LIN {X 0,Y 466.916,Z 269.289,A -85,B 0,C 180,E1 -7460.907,E2 -7460.907} C_VEL
LIN {X 0,Y 467.076,Z 265.162,A -85,B 0,C 180,E1 -7462.217,E2 -7462.217} C_VEL
LIN {X 0,Y 467.331,Z 259.259,A -85,B 0,C 180,E1 -7463.655,E2 -7463.655} C_VEL
LIN {X 0,Y 467.652,Z 252.016,A -85,B 0,C 180,E1 -7465.043,E2 -7465.043} C_VEL
LIN {X 0,Y 467.969,Z 245.037,A -85,B 0,C 180,E1 -7466.125,E2 -7466.125} C_VEL
LIN {X 0,Y 468.397,Z 236.625,A -85,B 0,C 180,E1 -7467.205,E2 -7467.205} C_VEL
LIN {X 0,Y 468.875,Z 226.254,A -85,B 0,C 180,E1 -7468.282,E2 -7468.282} C_VEL
LIN {X 0,Y 469.414,Z 214.581,A -85,B 0,C 180,E1 -7469.25,E2 -7469.25} C_VEL
LIN {X 0,Y 469.811,Z 202.915,A -85,B 0,C 180,E1 -7470,E2 -7470} C_VEL
LIN {X 0,Y 470.165,Z 189.535,A -85,B 0,C 180,E1 -7470.643,E2 -7470.643} C_VEL
LIN {X 0,Y 470.404,Z 177.571,A -85,B 0,C 180,E1 -7471.044,E2 -7471.044} C_VEL
LIN {X 0,Y 470.627,Z 162.533,A -85,B 0,C 180,E1 -7471.337,E2 -7471.337} C_VEL
LIN {X 0,Y 471.101,Z 78.839,A -85,B 0,C 180,E1 -7472.624,E2 -7472.624} C_VEL
LIN {X 0,Y 468.46,Z 65.811,A -85,B 0,C 180,E1 -7472.929,E2 -7472.929} C_VEL
LIN {X 0,Y 468.526,Z 59.499,A -85,B 0,C 180,E1 -7474.302,E2 -7474.302} C_VEL
LIN {X 0,Y 467.789,Z 54.217,A -85,B 0,C 180,E1 -7475.496,E2 -7475.496} C_VEL
LIN {X 0,Y 467.755,Z 54.218,A -85,B 0,C 180,E1 -7477.772,E2 -7477.772} C_VEL
LIN {X 0,Y 467.657,Z 54.228,A -85,B 0,C 180,E1 -7481.266,E2 -7481.266} C_VEL
LIN {X 0,Y 467.617,Z 54.234,A -85,B 0,C 180,E1 -7483.915,E2 -7483.915} C_VEL
LIN {X 0,Y 467.597,Z 54.24,A -85,B 0,C 180,E1 -7486.593,E2 -7486.593} C_VEL
LIN {X 0,Y 467.628,Z 54.231,A -85,B 0,C 180,E1 -7489.308,E2 -7489.308} C_VEL
LIN {X 0,Y 467.54,Z 54.248,A -85,B 0,C 180,E1 -7492.074,E2 -7492.074} C_VEL
LIN {X 0,Y 467.591,Z 54.236,A -85,B 0,C 180,E1 -7494.888,E2 -7494.888} C_VEL
LIN {X 0,Y 467.625,Z 54.236,A -85,B 0,C 180,E1 -7497.769,E2 -7497.769} C_VEL
LIN {X 0,Y 467.573,Z 54.238,A -85,B 0,C 180,E1 -7501.045,E2 -7501.045} C_VEL
LIN {X 0,Y 467.595,Z 54.237,A -85,B 0,C 180,E1 -7504.242,E2 -7504.242} C_VEL
LIN {X 0,Y 467.554,Z 54.242,A -85,B 0,C 180,E1 -7507.186,E2 -7507.186} C_VEL
LIN {X 0,Y 467.582,Z 54.237,A -85,B 0,C 180,E1 -7510.264,E2 -7510.264} C_VEL
LIN {X 0,Y 467.591,Z 54.236,A -85,B 0,C 180,E1 -7512.567,E2 -7512.567} C_VEL
LIN {X 0,Y 467.57,Z 54.242,A -85,B 0,C 180,E1 -7515.052,E2 -7515.052} C_VEL
LIN {X 0,Y 467.593,Z 54.241,A -85,B 0,C 180,E1 -7517.44,E2 -7517.44} C_VEL
LIN {X 0,Y 467.586,Z 54.24,A -85,B 0,C 180,E1 -7520.855,E2 -7520.855} C_VEL
LIN {X 0,Y 467.564,Z 54.239,A -85,B 0,C 180,E1 -7524.261,E2 -7524.261} C_VEL
LIN {X 0,Y 467.585,Z 54.239,A -85,B 0,C 180,E1 -7527.321,E2 -7527.321} C_VEL
LIN {X 0,Y 467.574,Z 54.244,A -85,B 0,C 180,E1 -7530.667,E2 -7530.667} C_VEL
LIN {X 0,Y 467.62,Z 54.234,A -85,B 0,C 180,E1 -7533.199,E2 -7533.199} C_VEL
LIN {X 0,Y 467.596,Z 54.241,A -85,B 0,C 180,E1 -7536.468,E2 -7536.468} C_VEL
LIN {X 0,Y 467.626,Z 54.232,A -85,B 0,C 180,E1 -7539.777,E2 -7539.777} C_VEL
LIN {X 0,Y 467.61,Z 54.24,A -85,B 0,C 180,E1 -7542.506,E2 -7542.506} C_VEL
LIN {X 0,Y 467.609,Z 54.233,A -85,B 0,C 180,E1 -7545.196,E2 -7545.196} C_VEL
LIN {X 0,Y 467.659,Z 54.23,A -85,B 0,C 180,E1 -7547.854,E2 -7547.854} C_VEL
LIN {X 0,Y 467.683,Z 54.225,A -85,B 0,C 180,E1 -7551.357,E2 -7551.357} C_VEL
LIN {X 0,Y 467.739,Z 54.225,A -85,B 0,C 180,E1 -7553.962,E2 -7553.962} C_VEL
LIN {X 0,Y 467.86,Z 54.204,A -85,B 0,C 180,E1 -7557.417,E2 -7557.417} C_VEL
LIN {X 0,Y 467.884,Z 54.204,A -85,B 0,C 180,E1 -7560,E2 -7560} C_VEL
LIN {X 0,Y 467.86,Z 54.202,A -85,B 0,C 180,E1 -7562.583,E2 -7562.583} C_VEL
LIN {X 0,Y 467.735,Z 54.22,A -85,B 0,C 180,E1 -7566.037,E2 -7566.037} C_VEL
LIN {X 0,Y 467.672,Z 54.226,A -85,B 0,C 180,E1 -7568.643,E2 -7568.643} C_VEL
LIN {X 0,Y 467.658,Z 54.227,A -85,B 0,C 180,E1 -7572.145,E2 -7572.145} C_VEL
LIN {X 0,Y 467.641,Z 54.232,A -85,B 0,C 180,E1 -7575.695,E2 -7575.695} C_VEL
LIN {X 0,Y 467.615,Z 54.236,A -85,B 0,C 180,E1 -7578.763,E2 -7578.763} C_VEL
LIN {X 0,Y 467.582,Z 54.241,A -85,B 0,C 180,E1 -7581.268,E2 -7581.268} C_VEL
LIN {X 0,Y 467.57,Z 54.238,A -85,B 0,C 180,E1 -7583.943,E2 -7583.943} C_VEL
LIN {X 0,Y 467.592,Z 54.243,A -85,B 0,C 180,E1 -7586.802,E2 -7586.802} C_VEL
LIN {X 0,Y 467.555,Z 54.24,A -85,B 0,C 180,E1 -7589.738,E2 -7589.738} C_VEL
LIN {X 0,Y 467.585,Z 54.243,A -85,B 0,C 180,E1 -7592.758,E2 -7592.758} C_VEL
LIN {X 0,Y 467.555,Z 54.241,A -85,B 0,C 180,E1 -7595.889,E2 -7595.889} C_VEL
LIN {X 0,Y 467.562,Z 54.24,A -85,B 0,C 180,E1 -7599.147,E2 -7599.147} C_VEL
LIN {X 0,Y 467.588,Z 54.24,A -85,B 0,C 180,E1 -7602.567,E2 -7602.567} C_VEL
LIN {X 0,Y 467.568,Z 54.239,A -85,B 0,C 180,E1 -7605.052,E2 -7605.052} C_VEL
LIN {X 0,Y 467.591,Z 54.236,A -85,B 0,C 180,E1 -7607.44,E2 -7607.44} C_VEL
LIN {X 0,Y 467.584,Z 54.237,A -85,B 0,C 180,E1 -7610.855,E2 -7610.855} C_VEL
LIN {X 0,Y 467.562,Z 54.242,A -85,B 0,C 180,E1 -7614.261,E2 -7614.261} C_VEL
LIN {X 0,Y 467.584,Z 54.239,A -85,B 0,C 180,E1 -7617.321,E2 -7617.321} C_VEL
LIN {X 0,Y 467.572,Z 54.244,A -85,B 0,C 180,E1 -7620.667,E2 -7620.667} C_VEL
LIN {X 0,Y 467.676,Z 54.389,A -85,B 0,C 180,E1 -7623.354,E2 -7623.354} C_VEL
LIN {X 0,Y 469.823,Z 66.098,A -85,B 0,C 180,E1 -7625.425,E2 -7625.425} C_VEL
LIN {X 0,Y 469.23,Z 83.836,A -85,B 0,C 180,E1 -7628.347,E2 -7628.347} C_VEL
LIN {X 0,Y 468.388,Z 105.455,A -85,B 0,C 180,E1 -7631.859,E2 -7631.859} C_VEL
LIN {X 0,Y 468.15,Z 113.126,A -85,B 0,C 180,E1 -7633.08,E2 -7633.08} C_VEL
LIN {X 0,Y 470.944,Z 133.853,A -85,B 0,C 180,E1 -7633.492,E2 -7633.492} C_VEL
LIN {X 0,Y 470.258,Z 222.266,A -85,B 0,C 180,E1 -7634.866,E2 -7634.866} C_VEL
LIN {X 0,Y 469.891,Z 235.42,A -85,B 0,C 180,E1 -7635.242,E2 -7635.242} C_VEL
LIN {X 0,Y 469.45,Z 247.547,A -85,B 0,C 180,E1 -7635.754,E2 -7635.754} C_VEL
LIN {X 0,Y 468.991,Z 259.804,A -85,B 0,C 180,E1 -7636.458,E2 -7636.458} C_VEL
LIN {X 0,Y 468.419,Z 272.106,A -85,B 0,C 180,E1 -7637.382,E2 -7637.382} C_VEL
LIN {X 0,Y 467.948,Z 282.93,A -85,B 0,C 180,E1 -7638.412,E2 -7638.412} C_VEL
LIN {X 0,Y 467.455,Z 292.948,A -85,B 0,C 180,E1 -7639.606,E2 -7639.606} C_VEL
LIN {X 0,Y 467.129,Z 301.775,A -85,B 0,C 180,E1 -7640.91,E2 -7640.91} C_VEL
LIN {X 0,Y 466.89,Z 308.811,A -85,B 0,C 180,E1 -7642.214,E2 -7642.214} C_VEL
LIN {X 0,Y 466.702,Z 314.993,A -85,B 0,C 180,E1 -7643.661,E2 -7643.661} C_VEL
LIN {X 0,Y 466.746,Z 318.872,A -85,B 0,C 180,E1 -7644.816,E2 -7644.816} C_VEL
LIN {X 0,Y 466.659,Z 321.204,A -85,B 0,C 180,E1 -7645.681,E2 -7645.681} C_VEL
LIN {X 0,Y 466.747,Z 323.112,A -85,B 0,C 180,E1 -7646.547,E2 -7646.547} C_VEL
LIN {X 0,Y 466.71,Z 324.547,A -85,B 0,C 180,E1 -7647.41,E2 -7647.41} C_VEL
LIN {X 0,Y 466.698,Z 325.564,A -85,B 0,C 180,E1 -7648.274,E2 -7648.274} C_VEL
LIN {X 0,Y 466.626,Z 326.421,A -85,B 0,C 180,E1 -7650,E2 -7650} C_VEL
LIN {X 0,Y 466.638,Z 326.228,A -85,B 0,C 180,E1 -7650.863,E2 -7650.863} C_VEL
LIN {X 0,Y 466.699,Z 325.63,A -85,B 0,C 180,E1 -7651.726,E2 -7651.726} C_VEL
LIN {X 0,Y 466.747,Z 323.253,A -85,B 0,C 180,E1 -7653.453,E2 -7653.453} C_VEL
LIN {X 0,Y 466.687,Z 320.32,A -85,B 0,C 180,E1 -7654.751,E2 -7654.751} C_VEL
LIN {X 0,Y 466.705,Z 316.357,A -85,B 0,C 180,E1 -7656.051,E2 -7656.051} C_VEL
LIN {X 0,Y 466.852,Z 311.265,A -85,B 0,C 180,E1 -7657.351,E2 -7657.351} C_VEL
LIN {X 0,Y 467.058,Z 304.877,A -85,B 0,C 180,E1 -7658.654,E2 -7658.654} C_VEL
LIN {X 0,Y 467.345,Z 296.895,A -85,B 0,C 180,E1 -7659.958,E2 -7659.958} C_VEL
LIN {X 0,Y 467.909,Z 286.997,A -85,B 0,C 180,E1 -7661.26,E2 -7661.26} C_VEL
LIN {X 0,Y 468.353,Z 277.342,A -85,B 0,C 180,E1 -7662.283,E2 -7662.283} C_VEL
LIN {X 0,Y 468.86,Z 266.461,A -85,B 0,C 180,E1 -7663.214,E2 -7663.214} C_VEL
LIN {X 0,Y 469.381,Z 255.345,A -85,B 0,C 180,E1 -7663.971,E2 -7663.971} C_VEL
LIN {X 0,Y 469.923,Z 243.021,A -85,B 0,C 180,E1 -7664.618,E2 -7664.618} C_VEL
LIN {X 0,Y 470.389,Z 229.964,A -85,B 0,C 180,E1 -7665.101,E2 -7665.101} C_VEL
LIN {X 0,Y 470.746,Z 217.491,A -85,B 0,C 180,E1 -7665.394,E2 -7665.394} C_VEL
LIN {X 0,Y 471.212,Z 132.613,A -85,B 0,C 180,E1 -7666.72,E2 -7666.72} C_VEL
LIN {X 0,Y 468.272,Z 112.505,A -85,B 0,C 180,E1 -7667.179,E2 -7667.179} C_VEL
LIN {X 0,Y 469.028,Z 94.371,A -85,B 0,C 180,E1 -7670.159,E2 -7670.159} C_VEL
LIN {X 0,Y 469.915,Z 73.905,A -85,B 0,C 180,E1 -7673.582,E2 -7673.582} C_VEL
LIN {X 0,Y 470.199,Z 67.087,A -85,B 0,C 180,E1 -7674.74,E2 -7674.74} C_VEL
LIN {X 0,Y 468.38,Z 57.447,A -85,B 0,C 180,E1 -7676.524,E2 -7676.524} C_VEL
LIN {X 0,Y 467.69,Z 54.229,A -85,B 0,C 180,E1 -7677.16,E2 -7677.16} C_VEL
LIN {X 0,Y 467.569,Z 54.245,A -85,B 0,C 180,E1 -7680.733,E2 -7680.733} C_VEL
LIN {X 0,Y 467.584,Z 54.244,A -85,B 0,C 180,E1 -7683.788,E2 -7683.788} C_VEL
LIN {X 0,Y 467.55,Z 54.243,A -85,B 0,C 180,E1 -7687.186,E2 -7687.186} C_VEL
LIN {X 0,Y 467.576,Z 54.242,A -85,B 0,C 180,E1 -7690.264,E2 -7690.264} C_VEL
LIN {X 0,Y 467.585,Z 54.238,A -85,B 0,C 180,E1 -7692.567,E2 -7692.567} C_VEL
LIN {X 0,Y 467.564,Z 54.239,A -85,B 0,C 180,E1 -7695.052,E2 -7695.052} C_VEL
LIN {X 0,Y 467.587,Z 54.241,A -85,B 0,C 180,E1 -7697.44,E2 -7697.44} C_VEL
LIN {X 0,Y 467.614,Z 54.235,A -85,B 0,C 180,E1 -7700.858,E2 -7700.858} C_VEL
LIN {X 0,Y 467.561,Z 54.24,A -85,B 0,C 180,E1 -7704.26,E2 -7704.26} C_VEL
LIN {X 0,Y 467.58,Z 54.243,A -85,B 0,C 180,E1 -7707.321,E2 -7707.321} C_VEL
LIN {X 0,Y 467.568,Z 54.242,A -85,B 0,C 180,E1 -7710.667,E2 -7710.667} C_VEL
LIN {X 0,Y 467.614,Z 54.234,A -85,B 0,C 180,E1 -7713.2,E2 -7713.2} C_VEL
LIN {X 0,Y 467.591,Z 54.241,A -85,B 0,C 180,E1 -7716.468,E2 -7716.468} C_VEL
LIN {X 0,Y 467.622,Z 54.233,A -85,B 0,C 180,E1 -7719.777,E2 -7719.777} C_VEL
LIN {X 0,Y 467.607,Z 54.235,A -85,B 0,C 180,E1 -7722.507,E2 -7722.507} C_VEL
LIN {X 0,Y 467.603,Z 54.235,A -85,B 0,C 180,E1 -7725.196,E2 -7725.196} C_VEL
LIN {X 0,Y 467.653,Z 54.225,A -85,B 0,C 180,E1 -7727.855,E2 -7727.855} C_VEL
LIN {X 0,Y 467.679,Z 54.224,A -85,B 0,C 180,E1 -7731.357,E2 -7731.357} C_VEL
LIN {X 0,Y 467.735,Z 54.222,A -85,B 0,C 180,E1 -7733.963,E2 -7733.963} C_VEL
LIN {X 0,Y 467.856,Z 54.203,A -85,B 0,C 180,E1 -7737.417,E2 -7737.417} C_VEL
LIN {X 0,Y 467.879,Z 54.205,A -85,B 0,C 180,E1 -7740,E2 -7740} C_VEL
LIN {X 0,Y 467.856,Z 54.198,A -85,B 0,C 180,E1 -7742.583,E2 -7742.583} C_VEL
LIN {X 0,Y 467.731,Z 54.22,A -85,B 0,C 180,E1 -7746.038,E2 -7746.038} C_VEL
LIN {X 0,Y 467.668,Z 54.222,A -85,B 0,C 180,E1 -7748.643,E2 -7748.643} C_VEL
LIN {X 0,Y 467.654,Z 54.226,A -85,B 0,C 180,E1 -7752.146,E2 -7752.146} C_VEL
LIN {X 0,Y 467.637,Z 54.231,A -85,B 0,C 180,E1 -7755.695,E2 -7755.695} C_VEL
LIN {X 0,Y 467.611,Z 54.236,A -85,B 0,C 180,E1 -7758.763,E2 -7758.763} C_VEL
LIN {X 0,Y 467.579,Z 54.236,A -85,B 0,C 180,E1 -7761.269,E2 -7761.269} C_VEL
LIN {X 0,Y 467.562,Z 54.241,A -85,B 0,C 180,E1 -7763.944,E2 -7763.944} C_VEL
LIN {X 0,Y 467.564,Z 54.245,A -85,B 0,C 180,E1 -7766.804,E2 -7766.804} C_VEL
LIN {X 0,Y 467.546,Z 54.24,A -85,B 0,C 180,E1 -7769.739,E2 -7769.739} C_VEL
LIN {X 0,Y 467.578,Z 54.241,A -85,B 0,C 180,E1 -7772.759,E2 -7772.759} C_VEL
LIN {X 0,Y 467.549,Z 54.243,A -85,B 0,C 180,E1 -7775.891,E2 -7775.891} C_VEL
LIN {X 0,Y 467.551,Z 54.244,A -85,B 0,C 180,E1 -7779.148,E2 -7779.148} C_VEL
LIN {X 0,Y 467.564,Z 54.237,A -85,B 0,C 180,E1 -7781.405,E2 -7781.405} C_VEL
LIN {X 0,Y 467.565,Z 54.239,A -85,B 0,C 180,E1 -7785.053,E2 -7785.053} C_VEL
LIN {X 0,Y 467.565,Z 54.24,A -85,B 0,C 180,E1 -7788.726,E2 -7788.726} C_VEL
LIN {X 0,Y 467.547,Z 54.248,A -85,B 0,C 180,E1 -7791.954,E2 -7791.954} C_VEL
LIN {X 0,Y 467.557,Z 54.249,A -85,B 0,C 180,E1 -7795.167,E2 -7795.167} C_VEL
LIN {X 0,Y 467.605,Z 54.347,A -85,B 0,C 180,E1 -7796.186,E2 -7796.186} C_VEL
LIN {X 0,Y 468.85,Z 61.426,A -85,B 0,C 180,E1 -7797.85,E2 -7797.85} C_VEL
LIN {X 0,Y 468.805,Z 66.288,A -85,B 0,C 180,E1 -7798.924,E2 -7798.924} C_VEL
LIN {X 0,Y 471.832,Z 79.918,A -85,B 0,C 180,E1 -7799.269,E2 -7799.269} C_VEL
LIN {X 0,Y 470.938,Z 172.284,A -85,B 0,C 180,E1 -7800.712,E2 -7800.712} C_VEL
LIN {X 0,Y 470.743,Z 183.575,A -85,B 0,C 180,E1 -7801.021,E2 -7801.021} C_VEL
LIN {X 0,Y 469.895,Z 189.287,A -85,B 0,C 180,E1 -7801.202,E2 -7801.202} C_VEL
LIN {X 0,Y 465.53,Z 201.989,A -85,B 0,C 180,E1 -7801.65,E2 -7801.65} C_VEL
LIN {X 0,Y 463.438,Z 209.017,A -85,B 0,C 180,E1 -7802.003,E2 -7802.003} C_VEL
LIN {X 0,Y 463.007,Z 212.433,A -85,B 0,C 180,E1 -7802.226,E2 -7802.226} C_VEL
LIN {X 0,Y 462.443,Z 223.732,A -85,B 0,C 180,E1 -7803.12,E2 -7803.12} C_VEL
LIN {X 0,Y 461.959,Z 233.267,A -85,B 0,C 180,E1 -7804.063,E2 -7804.063} C_VEL
LIN {X 0,Y 461.391,Z 242.873,A -85,B 0,C 180,E1 -7805.236,E2 -7805.236} C_VEL
LIN {X 0,Y 460.939,Z 250.637,A -85,B 0,C 180,E1 -7806.398,E2 -7806.398} C_VEL
LIN {X 0,Y 460.489,Z 258.274,A -85,B 0,C 180,E1 -7807.807,E2 -7807.807} C_VEL
LIN {X 0,Y 460.247,Z 263.603,A -85,B 0,C 180,E1 -7809.043,E2 -7809.043} C_VEL
LIN {X 0,Y 460.05,Z 268.129,A -85,B 0,C 180,E1 -7810.362,E2 -7810.362} C_VEL
LIN {X 0,Y 459.871,Z 270.811,A -85,B 0,C 180,E1 -7811.357,E2 -7811.357} C_VEL
LIN {X 0,Y 459.657,Z 274.227,A -85,B 0,C 180,E1 -7813.112,E2 -7813.112} C_VEL
LIN {X 0,Y 459.619,Z 275.682,A -85,B 0,C 180,E1 -7814.437,E2 -7814.437} C_VEL
LIN {X 0,Y 459.56,Z 276.252,A -85,B 0,C 180,E1 -7815.837,E2 -7815.837} C_VEL
LIN {X 0,Y 459.59,Z 276.094,A -85,B 0,C 180,E1 -7816.74,E2 -7816.74} C_VEL
LIN {X 0,Y 459.679,Z 275.066,A -85,B 0,C 180,E1 -7818.098,E2 -7818.098} C_VEL
LIN {X 0,Y 459.712,Z 273.122,A -85,B 0,C 180,E1 -7819.429,E2 -7819.429} C_VEL
LIN {X 0,Y 459.812,Z 270.194,A -85,B 0,C 180,E1 -7820.765,E2 -7820.765} C_VEL
LIN {X 0,Y 459.995,Z 266.224,A -85,B 0,C 180,E1 -7822.097,E2 -7822.097} C_VEL
LIN {X 0,Y 460.259,Z 260.296,A -85,B 0,C 180,E1 -7823.605,E2 -7823.605} C_VEL
LIN {X 0,Y 460.547,Z 253.46,A -85,B 0,C 180,E1 -7824.966,E2 -7824.966} C_VEL
LIN {X 0,Y 460.967,Z 245.209,A -85,B 0,C 180,E1 -7826.285,E2 -7826.285} C_VEL
LIN {X 0,Y 461.429,Z 236.726,A -85,B 0,C 180,E1 -7827.381,E2 -7827.381} C_VEL
LIN {X 0,Y 461.914,Z 226.288,A -85,B 0,C 180,E1 -7828.475,E2 -7828.475} C_VEL
LIN {X 0,Y 462.427,Z 215.936,A -85,B 0,C 180,E1 -7829.347,E2 -7829.347} C_VEL
LIN {X 0,Y 462.863,Z 204.608,A -85,B 0,C 180,E1 -7830.109,E2 -7830.109} C_VEL
LIN {X 0,Y 463.241,Z 191.654,A -85,B 0,C 180,E1 -7830.761,E2 -7830.761} C_VEL
LIN {X 0,Y 463.48,Z 179.532,A -85,B 0,C 180,E1 -7831.195,E2 -7831.195} C_VEL
LIN {X 0,Y 463.668,Z 166.043,A -85,B 0,C 180,E1 -7831.493,E2 -7831.493} C_VEL
LIN {X 0,Y 464.364,Z 80.659,A -85,B 0,C 180,E1 -7832.82,E2 -7832.82} C_VEL
LIN {X 0,Y 461.461,Z 66.202,A -85,B 0,C 180,E1 -7833.153,E2 -7833.153} C_VEL
LIN {X 0,Y 461.55,Z 60.66,A -85,B 0,C 180,E1 -7834.367,E2 -7834.367} C_VEL
LIN {X 0,Y 460.751,Z 55.093,A -85,B 0,C 180,E1 -7835.663,E2 -7835.663} C_VEL
LIN {X 0,Y 460.701,Z 55.098,A -85,B 0,C 180,E1 -7837.892,E2 -7837.892} C_VEL
LIN {X 0,Y 460.616,Z 55.104,A -85,B 0,C 180,E1 -7841.441,E2 -7841.441} C_VEL
LIN {X 0,Y 460.571,Z 55.111,A -85,B 0,C 180,E1 -7845.035,E2 -7845.035} C_VEL
LIN {X 0,Y 460.555,Z 55.114,A -85,B 0,C 180,E1 -7847.77,E2 -7847.77} C_VEL
LIN {X 0,Y 460.557,Z 55.116,A -85,B 0,C 180,E1 -7850.547,E2 -7850.547} C_VEL
LIN {X 0,Y 460.537,Z 55.117,A -85,B 0,C 180,E1 -7853.704,E2 -7853.704} C_VEL
LIN {X 0,Y 460.561,Z 55.116,A -85,B 0,C 180,E1 -7856.266,E2 -7856.266} C_VEL
LIN {X 0,Y 460.544,Z 55.114,A -85,B 0,C 180,E1 -7859.231,E2 -7859.231} C_VEL
LIN {X 0,Y 460.537,Z 55.117,A -85,B 0,C 180,E1 -7862.284,E2 -7862.284} C_VEL
LIN {X 0,Y 460.518,Z 55.121,A -85,B 0,C 180,E1 -7865.445,E2 -7865.445} C_VEL
LIN {X 0,Y 460.549,Z 55.114,A -85,B 0,C 180,E1 -7868.898,E2 -7868.898} C_VEL
LIN {X 0,Y 460.527,Z 55.116,A -85,B 0,C 180,E1 -7872.181,E2 -7872.181} C_VEL
LIN {X 0,Y 460.518,Z 55.124,A -85,B 0,C 180,E1 -7875.411,E2 -7875.411} C_VEL
LIN {X 0,Y 460.536,Z 55.115,A -85,B 0,C 180,E1 -7878.397,E2 -7878.397} C_VEL
LIN {X 0,Y 460.53,Z 55.121,A -85,B 0,C 180,E1 -7881.267,E2 -7881.267} C_VEL
LIN {X 0,Y 460.514,Z 55.119,A -85,B 0,C 180,E1 -7884.554,E2 -7884.554} C_VEL
LIN {X 0,Y 460.535,Z 55.115,A -85,B 0,C 180,E1 -7887.715,E2 -7887.715} C_VEL
LIN {X 0,Y 460.544,Z 55.121,A -85,B 0,C 180,E1 -7890.769,E2 -7890.769} C_VEL
LIN {X 0,Y 460.566,Z 55.111,A -85,B 0,C 180,E1 -7893.735,E2 -7893.735} C_VEL
LIN {X 0,Y 460.549,Z 55.121,A -85,B 0,C 180,E1 -7896.624,E2 -7896.624} C_VEL
LIN {X 0,Y 460.554,Z 55.112,A -85,B 0,C 180,E1 -7899.453,E2 -7899.453} C_VEL
LIN {X 0,Y 460.561,Z 55.117,A -85,B 0,C 180,E1 -7902.23,E2 -7902.23} C_VEL
LIN {X 0,Y 460.568,Z 55.111,A -85,B 0,C 180,E1 -7904.965,E2 -7904.965} C_VEL
LIN {X 0,Y 460.613,Z 55.108,A -85,B 0,C 180,E1 -7908.559,E2 -7908.559} C_VEL
LIN {X 0,Y 460.698,Z 55.102,A -85,B 0,C 180,E1 -7912.108,E2 -7912.108} C_VEL
LIN {X 0,Y 460.697,Z 55.095,A -85,B 0,C 180,E1 -7914.748,E2 -7914.748} C_VEL
LIN {X 0,Y 460.801,Z 55.083,A -85,B 0,C 180,E1 -7917.377,E2 -7917.377} C_VEL
LIN {X 0,Y 460.854,Z 55.08,A -85,B 0,C 180,E1 -7920,E2 -7920} C_VEL
LIN {X 0,Y 460.801,Z 55.081,A -85,B 0,C 180,E1 -7922.622,E2 -7922.622} C_VEL
LIN {X 0,Y 460.7,Z 55.095,A -85,B 0,C 180,E1 -7926.13,E2 -7926.13} C_VEL
LIN {X 0,Y 460.622,Z 55.104,A -85,B 0,C 180,E1 -7928.776,E2 -7928.776} C_VEL
LIN {X 0,Y 460.616,Z 55.104,A -85,B 0,C 180,E1 -7932.445,E2 -7932.445} C_VEL
LIN {X 0,Y 460.602,Z 55.106,A -85,B 0,C 180,E1 -7935.997,E2 -7935.997} C_VEL
LIN {X 0,Y 460.57,Z 55.112,A -85,B 0,C 180,E1 -7939.615,E2 -7939.615} C_VEL
LIN {X 0,Y 460.512,Z 55.119,A -85,B 0,C 180,E1 -7942.429,E2 -7942.429} C_VEL
LIN {X 0,Y 460.55,Z 55.113,A -85,B 0,C 180,E1 -7945.797,E2 -7945.797} C_VEL
LIN {X 0,Y 460.551,Z 55.114,A -85,B 0,C 180,E1 -7948.233,E2 -7948.233} C_VEL
LIN {X 0,Y 460.523,Z 55.117,A -85,B 0,C 180,E1 -7951.283,E2 -7951.283} C_VEL
LIN {X 0,Y 460.533,Z 55.122,A -85,B 0,C 180,E1 -7954.505,E2 -7954.505} C_VEL
LIN {X 0,Y 460.503,Z 55.119,A -85,B 0,C 180,E1 -7957.623,E2 -7957.623} C_VEL
LIN {X 0,Y 460.541,Z 55.12,A -85,B 0,C 180,E1 -7960.269,E2 -7960.269} C_VEL
LIN {X 0,Y 460.498,Z 55.119,A -85,B 0,C 180,E1 -7963.376,E2 -7963.376} C_VEL
LIN {X 0,Y 460.498,Z 55.121,A -85,B 0,C 180,E1 -7966.624,E2 -7966.624} C_VEL
LIN {X 0,Y 460.544,Z 55.117,A -85,B 0,C 180,E1 -7969.73,E2 -7969.73} C_VEL
LIN {X 0,Y 460.501,Z 55.12,A -85,B 0,C 180,E1 -7972.524,E2 -7972.524} C_VEL
LIN {X 0,Y 460.549,Z 55.118,A -85,B 0,C 180,E1 -7975.624,E2 -7975.624} C_VEL
LIN {X 0,Y 460.539,Z 55.114,A -85,B 0,C 180,E1 -7978.744,E2 -7978.744} C_VEL
LIN {X 0,Y 460.584,Z 55.116,A -85,B 0,C 180,E1 -7982.254,E2 -7982.254} C_VEL
LIN {X 0,Y 460.642,Z 55.195,A -85,B 0,C 180,E1 -7983.159,E2 -7983.159} C_VEL
LIN {X 0,Y 462.889,Z 67.415,A -85,B 0,C 180,E1 -7985.356,E2 -7985.356} C_VEL
LIN {X 0,Y 462.112,Z 86.808,A -85,B 0,C 180,E1 -7988.592,E2 -7988.592} C_VEL
LIN {X 0,Y 461.363,Z 106.289,A -85,B 0,C 180,E1 -7991.803,E2 -7991.803} C_VEL
LIN {X 0,Y 461.13,Z 112.601,A -85,B 0,C 180,E1 -7992.836,E2 -7992.836} C_VEL
LIN {X 0,Y 464.07,Z 135.367,A -85,B 0,C 180,E1 -7993.297,E2 -7993.297} C_VEL
LIN {X 0,Y 463.357,Z 221.938,A -85,B 0,C 180,E1 -7994.663,E2 -7994.663} C_VEL
LIN {X 0,Y 462.977,Z 235.088,A -85,B 0,C 180,E1 -7995.045,E2 -7995.045} C_VEL
LIN {X 0,Y 462.496,Z 247.782,A -85,B 0,C 180,E1 -7995.591,E2 -7995.591} C_VEL
LIN {X 0,Y 462.028,Z 259.069,A -85,B 0,C 180,E1 -7996.25,E2 -7996.25} C_VEL
LIN {X 0,Y 461.496,Z 270.047,A -85,B 0,C 180,E1 -7997.069,E2 -7997.069} C_VEL
LIN {X 0,Y 460.94,Z 281.29,A -85,B 0,C 180,E1 -7998.121,E2 -7998.121} C_VEL
LIN {X 0,Y 460.544,Z 290.756,A -85,B 0,C 180,E1 -7999.226,E2 -7999.226} C_VEL
LIN {X 0,Y 460.118,Z 299.888,A -85,B 0,C 180,E1 -8000.549,E2 -8000.549} C_VEL
LIN {X 0,Y 459.884,Z 307.251,A -85,B 0,C 180,E1 -8001.873,E2 -8001.873} C_VEL
LIN {X 0,Y 459.733,Z 312.232,A -85,B 0,C 180,E1 -8002.975,E2 -8002.975} C_VEL
LIN {X 0,Y 459.621,Z 317.066,A -85,B 0,C 180,E1 -8004.296,E2 -8004.296} C_VEL
LIN {X 0,Y 459.574,Z 320.767,A -85,B 0,C 180,E1 -8005.614,E2 -8005.614} C_VEL
LIN {X 0,Y 459.657,Z 322.684,A -85,B 0,C 180,E1 -8006.493,E2 -8006.493} C_VEL
LIN {X 0,Y 459.631,Z 324.136,A -85,B 0,C 180,E1 -8007.371,E2 -8007.371} C_VEL
LIN {X 0,Y 459.635,Z 325.162,A -85,B 0,C 180,E1 -8008.247,E2 -8008.247} C_VEL
LIN {X 0,Y 459.556,Z 326.034,A -85,B 0,C 180,E1 -8010,E2 -8010} C_VEL
LIN {X 0,Y 459.57,Z 325.856,A -85,B 0,C 180,E1 -8010.876,E2 -8010.876} C_VEL
LIN {X 0,Y 459.606,Z 325.264,A -85,B 0,C 180,E1 -8011.752,E2 -8011.752} C_VEL
LIN {X 0,Y 459.63,Z 324.281,A -85,B 0,C 180,E1 -8012.629,E2 -8012.629} C_VEL
LIN {X 0,Y 459.64,Z 322.9,A -85,B 0,C 180,E1 -8013.506,E2 -8013.506} C_VEL
LIN {X 0,Y 459.613,Z 319.983,A -85,B 0,C 180,E1 -8014.824,E2 -8014.824} C_VEL
LIN {X 0,Y 459.634,Z 315.362,A -85,B 0,C 180,E1 -8016.342,E2 -8016.342} C_VEL
LIN {X 0,Y 459.861,Z 308.974,A -85,B 0,C 180,E1 -8017.906,E2 -8017.906} C_VEL
LIN {X 0,Y 460.066,Z 302.122,A -85,B 0,C 180,E1 -8019.23,E2 -8019.23} C_VEL
LIN {X 0,Y 460.468,Z 293.629,A -85,B 0,C 180,E1 -8020.553,E2 -8020.553} C_VEL
LIN {X 0,Y 460.98,Z 284.909,A -85,B 0,C 180,E1 -8021.654,E2 -8021.654} C_VEL
LIN {X 0,Y 461.531,Z 273.823,A -85,B 0,C 180,E1 -8022.791,E2 -8022.791} C_VEL
LIN {X 0,Y 462.121,Z 263.567,A -85,B 0,C 180,E1 -8023.634,E2 -8023.634} C_VEL
LIN {X 0,Y 462.661,Z 251.718,A -85,B 0,C 180,E1 -8024.403,E2 -8024.403} C_VEL
LIN {X 0,Y 463.252,Z 239.425,A -85,B 0,C 180,E1 -8025.002,E2 -8025.002} C_VEL
LIN {X 0,Y 463.731,Z 226.859,A -85,B 0,C 180,E1 -8025.436,E2 -8025.436} C_VEL
LIN {X 0,Y 463.962,Z 213.966,A -85,B 0,C 180,E1 -8025.71,E2 -8025.71} C_VEL
LIN {X 0,Y 464.636,Z 134.861,A -85,B 0,C 180,E1 -8026.951,E2 -8026.951} C_VEL
LIN {X 0,Y 461.857,Z 115.48,A -85,B 0,C 180,E1 -8027.38,E2 -8027.38} C_VEL
LIN {X 0,Y 461.325,Z 112.145,A -85,B 0,C 180,E1 -8027.471,E2 -8027.471} C_VEL
LIN {X 0,Y 462.091,Z 94.192,A -85,B 0,C 180,E1 -8030.475,E2 -8030.475} C_VEL
LIN {X 0,Y 463.114,Z 73.76,A -85,B 0,C 180,E1 -8033.95,E2 -8033.95} C_VEL
LIN {X 0,Y 463.247,Z 68.116,A -85,B 0,C 180,E1 -8034.933,E2 -8034.933} C_VEL
LIN {X 0,Y 460.815,Z 56.062,A -85,B 0,C 180,E1 -8037.228,E2 -8037.228} C_VEL
LIN {X 0,Y 460.625,Z 55.109,A -85,B 0,C 180,E1 -8037.449,E2 -8037.449} C_VEL
LIN {X 0,Y 460.511,Z 55.126,A -85,B 0,C 180,E1 -8040.24,E2 -8040.24} C_VEL
LIN {X 0,Y 460.527,Z 55.12,A -85,B 0,C 180,E1 -8043.325,E2 -8043.325} C_VEL
LIN {X 0,Y 460.478,Z 55.126,A -85,B 0,C 180,E1 -8046.529,E2 -8046.529} C_VEL
LIN {X 0,Y 460.557,Z 55.119,A -85,B 0,C 180,E1 -8049.859,E2 -8049.859} C_VEL
LIN {X 0,Y 460.511,Z 55.119,A -85,B 0,C 180,E1 -8052.9,E2 -8052.9} C_VEL
LIN {X 0,Y 460.507,Z 55.116,A -85,B 0,C 180,E1 -8055.83,E2 -8055.83} C_VEL
LIN {X 0,Y 460.537,Z 55.118,A -85,B 0,C 180,E1 -8058.989,E2 -8058.989} C_VEL
LIN {X 0,Y 460.542,Z 55.121,A -85,B 0,C 180,E1 -8061.269,E2 -8061.269} C_VEL
LIN {X 0,Y 460.512,Z 55.119,A -85,B 0,C 180,E1 -8064.554,E2 -8064.554} C_VEL
LIN {X 0,Y 460.529,Z 55.117,A -85,B 0,C 180,E1 -8067.715,E2 -8067.715} C_VEL
LIN {X 0,Y 460.538,Z 55.118,A -85,B 0,C 180,E1 -8070.769,E2 -8070.769} C_VEL
LIN {X 0,Y 460.561,Z 55.109,A -85,B 0,C 180,E1 -8073.735,E2 -8073.735} C_VEL
LIN {X 0,Y 460.544,Z 55.118,A -85,B 0,C 180,E1 -8076.624,E2 -8076.624} C_VEL
LIN {X 0,Y 460.55,Z 55.113,A -85,B 0,C 180,E1 -8079.453,E2 -8079.453} C_VEL
LIN {X 0,Y 460.557,Z 55.113,A -85,B 0,C 180,E1 -8082.23,E2 -8082.23} C_VEL
LIN {X 0,Y 460.563,Z 55.113,A -85,B 0,C 180,E1 -8084.965,E2 -8084.965} C_VEL
LIN {X 0,Y 460.609,Z 55.109,A -85,B 0,C 180,E1 -8088.559,E2 -8088.559} C_VEL
LIN {X 0,Y 460.693,Z 55.095,A -85,B 0,C 180,E1 -8092.109,E2 -8092.109} C_VEL
LIN {X 0,Y 460.693,Z 55.096,A -85,B 0,C 180,E1 -8094.748,E2 -8094.748} C_VEL
LIN {X 0,Y 460.797,Z 55.082,A -85,B 0,C 180,E1 -8097.378,E2 -8097.378} C_VEL
LIN {X 0,Y 460.849,Z 55.08,A -85,B 0,C 180,E1 -8100,E2 -8100} C_VEL
LIN {X 0,Y 460.797,Z 55.077,A -85,B 0,C 180,E1 -8102.623,E2 -8102.623} C_VEL
LIN {X 0,Y 460.696,Z 55.095,A -85,B 0,C 180,E1 -8106.13,E2 -8106.13} C_VEL
LIN {X 0,Y 460.618,Z 55.101,A -85,B 0,C 180,E1 -8108.777,E2 -8108.777} C_VEL
LIN {X 0,Y 460.611,Z 55.103,A -85,B 0,C 180,E1 -8112.445,E2 -8112.445} C_VEL
LIN {X 0,Y 460.598,Z 55.107,A -85,B 0,C 180,E1 -8115.998,E2 -8115.998} C_VEL
LIN {X 0,Y 460.566,Z 55.112,A -85,B 0,C 180,E1 -8119.616,E2 -8119.616} C_VEL
LIN {X 0,Y 460.509,Z 55.117,A -85,B 0,C 180,E1 -8122.429,E2 -8122.429} C_VEL
LIN {X 0,Y 460.547,Z 55.11,A -85,B 0,C 180,E1 -8125.797,E2 -8125.797} C_VEL
LIN {X 0,Y 460.525,Z 55.121,A -85,B 0,C 180,E1 -8128.235,E2 -8128.235} C_VEL
LIN {X 0,Y 460.519,Z 55.118,A -85,B 0,C 180,E1 -8131.283,E2 -8131.283} C_VEL
LIN {X 0,Y 460.521,Z 55.12,A -85,B 0,C 180,E1 -8134.504,E2 -8134.504} C_VEL
LIN {X 0,Y 460.497,Z 55.123,A -85,B 0,C 180,E1 -8137.624,E2 -8137.624} C_VEL
LIN {X 0,Y 460.518,Z 55.113,A -85,B 0,C 180,E1 -8141.013,E2 -8141.013} C_VEL
LIN {X 0,Y 460.511,Z 55.118,A -85,B 0,C 180,E1 -8144.59,E2 -8144.59} C_VEL
LIN {X 0,Y 460.491,Z 55.129,A -85,B 0,C 180,E1 -8147.816,E2 -8147.816} C_VEL
LIN {X 0,Y 460.511,Z 55.123,A -85,B 0,C 180,E1 -8150.136,E2 -8150.136} C_VEL
LIN {X 0,Y 460.467,Z 55.132,A -85,B 0,C 180,E1 -8153.47,E2 -8153.47} C_VEL
LIN {X 0,Y 460.562,Z 55.223,A -85,B 0,C 180,E1 -8155.956,E2 -8155.956} C_VEL
LIN {X 0,Y 461.93,Z 63.082,A -85,B 0,C 180,E1 -8157.826,E2 -8157.826} C_VEL
LIN {X 0,Y 461.938,Z 66.897,A -85,B 0,C 180,E1 -8158.63,E2 -8158.63} C_VEL
LIN {X 0,Y 465.085,Z 80.736,A -85,B 0,C 180,E1 -8158.995,E2 -8158.995} C_VEL
LIN {X 0,Y 464.185,Z 172.963,A -85,B 0,C 180,E1 -8160.462,E2 -8160.462} C_VEL
LIN {X 0,Y 463.93,Z 186.168,A -85,B 0,C 180,E1 -8160.848,E2 -8160.848} C_VEL
LIN {X 0,Y 463.585,Z 199.092,A -85,B 0,C 180,E1 -8161.414,E2 -8161.414} C_VEL
LIN {X 0,Y 463.133,Z 210.084,A -85,B 0,C 180,E1 -8162.062,E2 -8162.062} C_VEL
LIN {X 0,Y 463.007,Z 212.433,A -85,B 0,C 180,E1 -8162.226,E2 -8162.226} C_VEL
LIN {X 0,Y 462.15,Z 217.571,A -85,B 0,C 180,E1 -8162.581,E2 -8162.581} C_VEL
LIN {X 0,Y 458.965,Z 225.695,A -85,B 0,C 180,E1 -8163.173,E2 -8163.173} C_VEL
LIN {X 0,Y 455.745,Z 233.358,A -85,B 0,C 180,E1 -8163.842,E2 -8163.842} C_VEL
LIN {X 0,Y 454.807,Z 237.718,A -85,B 0,C 180,E1 -8164.322,E2 -8164.322} C_VEL
LIN {X 0,Y 454.29,Z 246.491,A -85,B 0,C 180,E1 -8165.503,E2 -8165.503} C_VEL
LIN {X 0,Y 453.784,Z 253.998,A -85,B 0,C 180,E1 -8166.739,E2 -8166.739} C_VEL
LIN {X 0,Y 453.351,Z 260.942,A -85,B 0,C 180,E1 -8168.158,E2 -8168.158} C_VEL
LIN {X 0,Y 453.11,Z 266.396,A -85,B 0,C 180,E1 -8169.575,E2 -8169.575} C_VEL
LIN {X 0,Y 452.827,Z 271.11,A -85,B 0,C 180,E1 -8171.217,E2 -8171.217} C_VEL
LIN {X 0,Y 452.596,Z 274.302,A -85,B 0,C 180,E1 -8172.841,E2 -8172.841} C_VEL
LIN {X 0,Y 452.529,Z 276.034,A -85,B 0,C 180,E1 -8174.344,E2 -8174.344} C_VEL
LIN {X 0,Y 452.489,Z 276.604,A -85,B 0,C 180,E1 -8175.611,E2 -8175.611} C_VEL
LIN {X 0,Y 452.485,Z 276.543,A -85,B 0,C 180,E1 -8176.528,E2 -8176.528} C_VEL
LIN {X 0,Y 452.589,Z 275.512,A -85,B 0,C 180,E1 -8178.042,E2 -8178.042} C_VEL
LIN {X 0,Y 452.637,Z 273.816,A -85,B 0,C 180,E1 -8179.262,E2 -8179.262} C_VEL
LIN {X 0,Y 452.721,Z 271.029,A -85,B 0,C 180,E1 -8180.619,E2 -8180.619} C_VEL
LIN {X 0,Y 452.907,Z 267.209,A -85,B 0,C 180,E1 -8181.972,E2 -8181.972} C_VEL
LIN {X 0,Y 453.121,Z 262.206,A -85,B 0,C 180,E1 -8183.336,E2 -8183.336} C_VEL
LIN {X 0,Y 453.427,Z 256.06,A -85,B 0,C 180,E1 -8184.664,E2 -8184.664} C_VEL
LIN {X 0,Y 453.785,Z 248.32,A -85,B 0,C 180,E1 -8186.004,E2 -8186.004} C_VEL
LIN {X 0,Y 454.337,Z 238.637,A -85,B 0,C 180,E1 -8187.341,E2 -8187.341} C_VEL
LIN {X 0,Y 454.877,Z 228.622,A -85,B 0,C 180,E1 -8188.451,E2 -8188.451} C_VEL
LIN {X 0,Y 455.438,Z 217.284,A -85,B 0,C 180,E1 -8189.448,E2 -8189.448} C_VEL
LIN {X 0,Y 455.909,Z 206.186,A -85,B 0,C 180,E1 -8190.221,E2 -8190.221} C_VEL
LIN {X 0,Y 456.27,Z 193.805,A -85,B 0,C 180,E1 -8190.883,E2 -8190.883} C_VEL
LIN {X 0,Y 456.569,Z 181.473,A -85,B 0,C 180,E1 -8191.351,E2 -8191.351} C_VEL
LIN {X 0,Y 456.782,Z 167.634,A -85,B 0,C 180,E1 -8191.681,E2 -8191.681} C_VEL
LIN {X 0,Y 457.471,Z 81.186,A -85,B 0,C 180,E1 -8193.046,E2 -8193.046} C_VEL
LIN {X 0,Y 454.529,Z 66.458,A -85,B 0,C 180,E1 -8193.408,E2 -8193.408} C_VEL
LIN {X 0,Y 454.568,Z 61.835,A -85,B 0,C 180,E1 -8194.434,E2 -8194.434} C_VEL
LIN {X 0,Y 453.71,Z 55.971,A -85,B 0,C 180,E1 -8195.835,E2 -8195.835} C_VEL
LIN {X 0,Y 453.658,Z 55.976,A -85,B 0,C 180,E1 -8198.015,E2 -8198.015} C_VEL
LIN {X 0,Y 453.565,Z 55.983,A -85,B 0,C 180,E1 -8201.621,E2 -8201.621} C_VEL
LIN {X 0,Y 453.546,Z 55.985,A -85,B 0,C 180,E1 -8205.274,E2 -8205.274} C_VEL
LIN {X 0,Y 453.51,Z 55.994,A -85,B 0,C 180,E1 -8208.056,E2 -8208.056} C_VEL
LIN {X 0,Y 453.488,Z 55.993,A -85,B 0,C 180,E1 -8210.882,E2 -8210.882} C_VEL
LIN {X 0,Y 453.5,Z 55.996,A -85,B 0,C 180,E1 -8213.887,E2 -8213.887} C_VEL
LIN {X 0,Y 453.507,Z 55.991,A -85,B 0,C 180,E1 -8216.706,E2 -8216.706} C_VEL
LIN {X 0,Y 453.48,Z 55.999,A -85,B 0,C 180,E1 -8219.732,E2 -8219.732} C_VEL
LIN {X 0,Y 453.496,Z 55.993,A -85,B 0,C 180,E1 -8223.189,E2 -8223.189} C_VEL
LIN {X 0,Y 453.46,Z 55.997,A -85,B 0,C 180,E1 -8226.299,E2 -8226.299} C_VEL
LIN {X 0,Y 453.521,Z 55.994,A -85,B 0,C 180,E1 -8229.447,E2 -8229.447} C_VEL
LIN {X 0,Y 453.467,Z 55.997,A -85,B 0,C 180,E1 -8232.995,E2 -8232.995} C_VEL
LIN {X 0,Y 453.467,Z 55.997,A -85,B 0,C 180,E1 -8235.779,E2 -8235.779} C_VEL
LIN {X 0,Y 453.483,Z 55.993,A -85,B 0,C 180,E1 -8238.209,E2 -8238.209} C_VEL
LIN {X 0,Y 453.498,Z 55.994,A -85,B 0,C 180,E1 -8240.793,E2 -8240.793} C_VEL
LIN {X 0,Y 453.458,Z 55.996,A -85,B 0,C 180,E1 -8243.917,E2 -8243.917} C_VEL
LIN {X 0,Y 453.486,Z 55.998,A -85,B 0,C 180,E1 -8247.151,E2 -8247.151} C_VEL
LIN {X 0,Y 453.478,Z 55.995,A -85,B 0,C 180,E1 -8250.268,E2 -8250.268} C_VEL
LIN {X 0,Y 453.51,Z 55.991,A -85,B 0,C 180,E1 -8253.294,E2 -8253.294} C_VEL
LIN {X 0,Y 453.507,Z 55.993,A -85,B 0,C 180,E1 -8256.239,E2 -8256.239} C_VEL
LIN {X 0,Y 453.485,Z 55.994,A -85,B 0,C 180,E1 -8259.117,E2 -8259.117} C_VEL
LIN {X 0,Y 453.514,Z 55.991,A -85,B 0,C 180,E1 -8261.944,E2 -8261.944} C_VEL
LIN {X 0,Y 453.543,Z 55.988,A -85,B 0,C 180,E1 -8264.726,E2 -8264.726} C_VEL
LIN {X 0,Y 453.562,Z 55.988,A -85,B 0,C 180,E1 -8268.379,E2 -8268.379} C_VEL
LIN {X 0,Y 453.655,Z 55.978,A -85,B 0,C 180,E1 -8271.985,E2 -8271.985} C_VEL
LIN {X 0,Y 453.67,Z 55.97,A -85,B 0,C 180,E1 -8274.667,E2 -8274.667} C_VEL
LIN {X 0,Y 453.745,Z 55.962,A -85,B 0,C 180,E1 -8277.336,E2 -8277.336} C_VEL
LIN {X 0,Y 453.824,Z 55.955,A -85,B 0,C 180,E1 -8280,E2 -8280} C_VEL
LIN {X 0,Y 453.745,Z 55.96,A -85,B 0,C 180,E1 -8282.663,E2 -8282.663} C_VEL
LIN {X 0,Y 453.668,Z 55.971,A -85,B 0,C 180,E1 -8286.225,E2 -8286.225} C_VEL
LIN {X 0,Y 453.588,Z 55.981,A -85,B 0,C 180,E1 -8288.913,E2 -8288.913} C_VEL
LIN {X 0,Y 453.566,Z 55.983,A -85,B 0,C 180,E1 -8292.529,E2 -8292.529} C_VEL
LIN {X 0,Y 453.546,Z 55.985,A -85,B 0,C 180,E1 -8296.196,E2 -8296.196} C_VEL
LIN {X 0,Y 453.519,Z 55.995,A -85,B 0,C 180,E1 -8299.039,E2 -8299.039} C_VEL
LIN {X 0,Y 453.478,Z 55.994,A -85,B 0,C 180,E1 -8301.836,E2 -8301.836} C_VEL
LIN {X 0,Y 453.505,Z 55.996,A -85,B 0,C 180,E1 -8304.735,E2 -8304.735} C_VEL
LIN {X 0,Y 453.53,Z 55.987,A -85,B 0,C 180,E1 -8307.959,E2 -8307.959} C_VEL
LIN {X 0,Y 453.467,Z 55.995,A -85,B 0,C 180,E1 -8311.525,E2 -8311.525} C_VEL
LIN {X 0,Y 453.489,Z 55.997,A -85,B 0,C 180,E1 -8314.777,E2 -8314.777} C_VEL
LIN {X 0,Y 453.462,Z 56.002,A -85,B 0,C 180,E1 -8318.312,E2 -8318.312} C_VEL
LIN {X 0,Y 453.495,Z 55.996,A -85,B 0,C 180,E1 -8320.609,E2 -8320.609} C_VEL
LIN {X 0,Y 453.454,Z 55.997,A -85,B 0,C 180,E1 -8323.244,E2 -8323.244} C_VEL
LIN {X 0,Y 453.464,Z 55.998,A -85,B 0,C 180,E1 -8325.778,E2 -8325.778} C_VEL
LIN {X 0,Y 453.481,Z 55.999,A -85,B 0,C 180,E1 -8328.209,E2 -8328.209} C_VEL
LIN {X 0,Y 453.496,Z 55.992,A -85,B 0,C 180,E1 -8330.793,E2 -8330.793} C_VEL
LIN {X 0,Y 453.457,Z 56.004,A -85,B 0,C 180,E1 -8333.917,E2 -8333.917} C_VEL
LIN {X 0,Y 453.485,Z 55.994,A -85,B 0,C 180,E1 -8337.151,E2 -8337.151} C_VEL
LIN {X 0,Y 453.477,Z 56.002,A -85,B 0,C 180,E1 -8340.268,E2 -8340.268} C_VEL
LIN {X 0,Y 453.614,Z 56.157,A -85,B 0,C 180,E1 -8342.99,E2 -8342.99} C_VEL
LIN {X 0,Y 455.856,Z 68.009,A -85,B 0,C 180,E1 -8345.158,E2 -8345.158} C_VEL
LIN {X 0,Y 455.465,Z 79.226,A -85,B 0,C 180,E1 -8347.069,E2 -8347.069} C_VEL
LIN {X 0,Y 454.746,Z 95.975,A -85,B 0,C 180,E1 -8349.887,E2 -8349.887} C_VEL
LIN {X 0,Y 454.114,Z 112.337,A -85,B 0,C 180,E1 -8352.604,E2 -8352.604} C_VEL
LIN {X 0,Y 457.214,Z 135.978,A -85,B 0,C 180,E1 -8353.086,E2 -8353.086} C_VEL
LIN {X 0,Y 456.457,Z 221.473,A -85,B 0,C 180,E1 -8354.454,E2 -8354.454} C_VEL
LIN {X 0,Y 456.066,Z 234.651,A -85,B 0,C 180,E1 -8354.841,E2 -8354.841} C_VEL
LIN {X 0,Y 455.58,Z 246.79,A -85,B 0,C 180,E1 -8355.368,E2 -8355.368} C_VEL
LIN {X 0,Y 455.07,Z 258.248,A -85,B 0,C 180,E1 -8356.036,E2 -8356.036} C_VEL
LIN {X 0,Y 454.506,Z 269.873,A -85,B 0,C 180,E1 -8356.915,E2 -8356.915} C_VEL
LIN {X 0,Y 453.943,Z 280.621,A -85,B 0,C 180,E1 -8357.935,E2 -8357.935} C_VEL
LIN {X 0,Y 453.53,Z 290.163,A -85,B 0,C 180,E1 -8359.057,E2 -8359.057} C_VEL
LIN {X 0,Y 453.073,Z 299.34,A -85,B 0,C 180,E1 -8360.401,E2 -8360.401} C_VEL
LIN {X 0,Y 452.813,Z 306.739,A -85,B 0,C 180,E1 -8361.745,E2 -8361.745} C_VEL
LIN {X 0,Y 452.657,Z 311.748,A -85,B 0,C 180,E1 -8362.865,E2 -8362.865} C_VEL
LIN {X 0,Y 452.525,Z 316.986,A -85,B 0,C 180,E1 -8364.324,E2 -8364.324} C_VEL
LIN {X 0,Y 452.494,Z 320.329,A -85,B 0,C 180,E1 -8365.546,E2 -8365.546} C_VEL
LIN {X 0,Y 452.553,Z 322.254,A -85,B 0,C 180,E1 -8366.438,E2 -8366.438} C_VEL
LIN {X 0,Y 452.553,Z 323.725,A -85,B 0,C 180,E1 -8367.329,E2 -8367.329} C_VEL
LIN {X 0,Y 452.543,Z 324.758,A -85,B 0,C 180,E1 -8368.22,E2 -8368.22} C_VEL
LIN {X 0,Y 452.488,Z 325.646,A -85,B 0,C 180,E1 -8370,E2 -8370} C_VEL
LIN {X 0,Y 452.504,Z 325.483,A -85,B 0,C 180,E1 -8370.89,E2 -8370.89} C_VEL
LIN {X 0,Y 452.552,Z 323.923,A -85,B 0,C 180,E1 -8372.67,E2 -8372.67} C_VEL
LIN {X 0,Y 452.536,Z 322.549,A -85,B 0,C 180,E1 -8373.561,E2 -8373.561} C_VEL
LIN {X 0,Y 452.539,Z 319.653,A -85,B 0,C 180,E1 -8374.9,E2 -8374.9} C_VEL
LIN {X 0,Y 452.553,Z 315.435,A -85,B 0,C 180,E1 -8376.331,E2 -8376.331} C_VEL
LIN {X 0,Y 452.719,Z 310.679,A -85,B 0,C 180,E1 -8377.582,E2 -8377.582} C_VEL
LIN {X 0,Y 452.923,Z 304.352,A -85,B 0,C 180,E1 -8378.926,E2 -8378.926} C_VEL
LIN {X 0,Y 453.281,Z 296.453,A -85,B 0,C 180,E1 -8380.271,E2 -8380.271} C_VEL
LIN {X 0,Y 453.83,Z 288.425,A -85,B 0,C 180,E1 -8381.387,E2 -8381.387} C_VEL
LIN {X 0,Y 454.327,Z 278.649,A -85,B 0,C 180,E1 -8382.507,E2 -8382.507} C_VEL
LIN {X 0,Y 454.935,Z 267.8,A -85,B 0,C 180,E1 -8383.512,E2 -8383.512} C_VEL
LIN {X 0,Y 455.536,Z 257.227,A -85,B 0,C 180,E1 -8384.291,E2 -8384.291} C_VEL
LIN {X 0,Y 456.19,Z 244.529,A -85,B 0,C 180,E1 -8385.011,E2 -8385.011} C_VEL
LIN {X 0,Y 456.699,Z 231.848,A -85,B 0,C 180,E1 -8385.537,E2 -8385.537} C_VEL
LIN {X 0,Y 457.161,Z 219.761,A -85,B 0,C 180,E1 -8385.864,E2 -8385.864} C_VEL
LIN {X 0,Y 457.76,Z 134.333,A -85,B 0,C 180,E1 -8387.249,E2 -8387.249} C_VEL
LIN {X 0,Y 454.779,Z 114.277,A -85,B 0,C 180,E1 -8387.71,E2 -8387.71} C_VEL
LIN {X 0,Y 454.366,Z 111.733,A -85,B 0,C 180,E1 -8387.784,E2 -8387.784} C_VEL
LIN {X 0,Y 455.142,Z 95.395,A -85,B 0,C 180,E1 -8390.566,E2 -8390.566} C_VEL
LIN {X 0,Y 456.237,Z 74.997,A -85,B 0,C 180,E1 -8394.092,E2 -8394.092} C_VEL
LIN {X 0,Y 456.352,Z 69.557,A -85,B 0,C 180,E1 -8395.056,E2 -8395.056} C_VEL
LIN {X 0,Y 453.901,Z 57.331,A -85,B 0,C 180,E1 -8397.428,E2 -8397.428} C_VEL
LIN {X 0,Y 453.546,Z 55.992,A -85,B 0,C 180,E1 -8397.701,E2 -8397.701} C_VEL
LIN {X 0,Y 453.476,Z 56,A -85,B 0,C 180,E1 -8400.759,E2 -8400.759} C_VEL
LIN {X 0,Y 453.476,Z 56.003,A -85,B 0,C 180,E1 -8403.912,E2 -8403.912} C_VEL
LIN {X 0,Y 453.47,Z 55.998,A -85,B 0,C 180,E1 -8407.187,E2 -8407.187} C_VEL
LIN {X 0,Y 453.516,Z 55.993,A -85,B 0,C 180,E1 -8409.447,E2 -8409.447} C_VEL
LIN {X 0,Y 453.461,Z 55.998,A -85,B 0,C 180,E1 -8412.995,E2 -8412.995} C_VEL
LIN {X 0,Y 453.462,Z 55.993,A -85,B 0,C 180,E1 -8415.778,E2 -8415.778} C_VEL
LIN {X 0,Y 453.514,Z 55.993,A -85,B 0,C 180,E1 -8419.405,E2 -8419.405} C_VEL
LIN {X 0,Y 453.475,Z 55.992,A -85,B 0,C 180,E1 -8422.222,E2 -8422.222} C_VEL
LIN {X 0,Y 453.487,Z 55.996,A -85,B 0,C 180,E1 -8425.222,E2 -8425.222} C_VEL
LIN {X 0,Y 453.464,Z 55.998,A -85,B 0,C 180,E1 -8428.475,E2 -8428.475} C_VEL
LIN {X 0,Y 453.535,Z 55.987,A -85,B 0,C 180,E1 -8432.039,E2 -8432.039} C_VEL
LIN {X 0,Y 453.512,Z 55.992,A -85,B 0,C 180,E1 -8435.266,E2 -8435.266} C_VEL
LIN {X 0,Y 453.478,Z 55.993,A -85,B 0,C 180,E1 -8438.415,E2 -8438.415} C_VEL
LIN {X 0,Y 453.52,Z 55.988,A -85,B 0,C 180,E1 -8441.009,E2 -8441.009} C_VEL
LIN {X 0,Y 453.566,Z 55.983,A -85,B 0,C 180,E1 -8443.88,E2 -8443.88} C_VEL
LIN {X 0,Y 453.561,Z 55.977,A -85,B 0,C 180,E1 -8447.471,E2 -8447.471} C_VEL
LIN {X 0,Y 453.59,Z 55.979,A -85,B 0,C 180,E1 -8451.087,E2 -8451.087} C_VEL
LIN {X 0,Y 453.669,Z 55.971,A -85,B 0,C 180,E1 -8453.775,E2 -8453.775} C_VEL
LIN {X 0,Y 453.741,Z 55.96,A -85,B 0,C 180,E1 -8457.337,E2 -8457.337} C_VEL
LIN {X 0,Y 453.82,Z 55.956,A -85,B 0,C 180,E1 -8460,E2 -8460} C_VEL
LIN {X 0,Y 453.741,Z 55.956,A -85,B 0,C 180,E1 -8462.664,E2 -8462.664} C_VEL
LIN {X 0,Y 453.663,Z 55.971,A -85,B 0,C 180,E1 -8466.226,E2 -8466.226} C_VEL
LIN {X 0,Y 453.584,Z 55.978,A -85,B 0,C 180,E1 -8468.914,E2 -8468.914} C_VEL
LIN {X 0,Y 453.561,Z 55.982,A -85,B 0,C 180,E1 -8472.529,E2 -8472.529} C_VEL
LIN {X 0,Y 453.542,Z 55.986,A -85,B 0,C 180,E1 -8476.196,E2 -8476.196} C_VEL
LIN {X 0,Y 453.516,Z 55.996,A -85,B 0,C 180,E1 -8479.04,E2 -8479.04} C_VEL
LIN {X 0,Y 453.475,Z 55.99,A -85,B 0,C 180,E1 -8481.837,E2 -8481.837} C_VEL
LIN {X 0,Y 453.5,Z 55.995,A -85,B 0,C 180,E1 -8484.736,E2 -8484.736} C_VEL
LIN {X 0,Y 453.505,Z 55.993,A -85,B 0,C 180,E1 -8487.954,E2 -8487.954} C_VEL
LIN {X 0,Y 453.474,Z 55.999,A -85,B 0,C 180,E1 -8490.76,E2 -8490.76} C_VEL
LIN {X 0,Y 453.467,Z 55.999,A -85,B 0,C 180,E1 -8493.914,E2 -8493.914} C_VEL
LIN {X 0,Y 453.448,Z 55.999,A -85,B 0,C 180,E1 -8497.191,E2 -8497.191} C_VEL
LIN {X 0,Y 453.47,Z 55.992,A -85,B 0,C 180,E1 -8500.612,E2 -8500.612} C_VEL
LIN {X 0,Y 453.459,Z 56,A -85,B 0,C 180,E1 -8504.223,E2 -8504.223} C_VEL
LIN {X 0,Y 453.437,Z 56.005,A -85,B 0,C 180,E1 -8507.003,E2 -8507.003} C_VEL
LIN {X 0,Y 453.471,Z 56.001,A -85,B 0,C 180,E1 -8509.413,E2 -8509.413} C_VEL
LIN {X 0,Y 453.44,Z 56.004,A -85,B 0,C 180,E1 -8512.81,E2 -8512.81} C_VEL
LIN {X 0,Y 453.532,Z 56.142,A -85,B 0,C 180,E1 -8515.724,E2 -8515.724} C_VEL
LIN {X 0,Y 455.012,Z 64.616,A -85,B 0,C 180,E1 -8517.772,E2 -8517.772} C_VEL
LIN {X 0,Y 455.028,Z 66.936,A -85,B 0,C 180,E1 -8518.303,E2 -8518.303} C_VEL
LIN {X 0,Y 458.344,Z 81.429,A -85,B 0,C 180,E1 -8518.705,E2 -8518.705} C_VEL
LIN {X 0,Y 457.444,Z 173.795,A -85,B 0,C 180,E1 -8520.204,E2 -8520.204} C_VEL
LIN {X 0,Y 457.18,Z 186.725,A -85,B 0,C 180,E1 -8520.592,E2 -8520.592} C_VEL
LIN {X 0,Y 456.827,Z 199.318,A -85,B 0,C 180,E1 -8521.153,E2 -8521.153} C_VEL
LIN {X 0,Y 456.283,Z 211.011,A -85,B 0,C 180,E1 -8521.855,E2 -8521.855} C_VEL
LIN {X 0,Y 455.713,Z 221.807,A -85,B 0,C 180,E1 -8522.69,E2 -8522.69} C_VEL
LIN {X 0,Y 455.137,Z 232.222,A -85,B 0,C 180,E1 -8523.696,E2 -8523.696} C_VEL
LIN {X 0,Y 454.807,Z 237.718,A -85,B 0,C 180,E1 -8524.322,E2 -8524.322} C_VEL
LIN {X 0,Y 453.881,Z 241.969,A -85,B 0,C 180,E1 -8524.828,E2 -8524.828} C_VEL
LIN {X 0,Y 450.642,Z 248.547,A -85,B 0,C 180,E1 -8525.676,E2 -8525.676} C_VEL
LIN {X 0,Y 447.45,Z 254.506,A -85,B 0,C 180,E1 -8526.602,E2 -8526.602} C_VEL
LIN {X 0,Y 446.609,Z 257.774,A -85,B 0,C 180,E1 -8527.223,E2 -8527.223} C_VEL
LIN {X 0,Y 446.209,Z 264.377,A -85,B 0,C 180,E1 -8528.761,E2 -8528.761} C_VEL
LIN {X 0,Y 445.96,Z 269.116,A -85,B 0,C 180,E1 -8530.195,E2 -8530.195} C_VEL
LIN {X 0,Y 445.676,Z 272.648,A -85,B 0,C 180,E1 -8531.616,E2 -8531.616} C_VEL
LIN {X 0,Y 445.539,Z 274.375,A -85,B 0,C 180,E1 -8532.56,E2 -8532.56} C_VEL
LIN {X 0,Y 445.444,Z 276.385,A -85,B 0,C 180,E1 -8534.246,E2 -8534.246} C_VEL
LIN {X 0,Y 445.406,Z 276.958,A -85,B 0,C 180,E1 -8535.377,E2 -8535.377} C_VEL
LIN {X 0,Y 445.407,Z 276.964,A -85,B 0,C 180,E1 -8536.31,E2 -8536.31} C_VEL
LIN {X 0,Y 445.512,Z 275.956,A -85,B 0,C 180,E1 -8537.978,E2 -8537.978} C_VEL
LIN {X 0,Y 445.548,Z 274.51,A -85,B 0,C 180,E1 -8539.089,E2 -8539.089} C_VEL
LIN {X 0,Y 445.638,Z 271.864,A -85,B 0,C 180,E1 -8540.469,E2 -8540.469} C_VEL
LIN {X 0,Y 445.821,Z 268.193,A -85,B 0,C 180,E1 -8541.844,E2 -8541.844} C_VEL
LIN {X 0,Y 446.052,Z 262.958,A -85,B 0,C 180,E1 -8543.328,E2 -8543.328} C_VEL
LIN {X 0,Y 446.387,Z 256.268,A -85,B 0,C 180,E1 -8544.806,E2 -8544.806} C_VEL
LIN {X 0,Y 446.775,Z 248.471,A -85,B 0,C 180,E1 -8546.167,E2 -8546.167} C_VEL
LIN {X 0,Y 447.262,Z 240.506,A -85,B 0,C 180,E1 -8547.298,E2 -8547.298} C_VEL
LIN {X 0,Y 447.831,Z 230.8,A -85,B 0,C 180,E1 -8548.427,E2 -8548.427} C_VEL
LIN {X 0,Y 448.411,Z 220.002,A -85,B 0,C 180,E1 -8549.439,E2 -8549.439} C_VEL
LIN {X 0,Y 448.957,Z 207.709,A -85,B 0,C 180,E1 -8550.337,E2 -8550.337} C_VEL
LIN {X 0,Y 449.332,Z 195.721,A -85,B 0,C 180,E1 -8551.009,E2 -8551.009} C_VEL
LIN {X 0,Y 449.635,Z 183.312,A -85,B 0,C 180,E1 -8551.512,E2 -8551.512} C_VEL
LIN {X 0,Y 449.877,Z 170.076,A -85,B 0,C 180,E1 -8551.852,E2 -8551.852} C_VEL
LIN {X 0,Y 450.633,Z 82.258,A -85,B 0,C 180,E1 -8553.265,E2 -8553.265} C_VEL
LIN {X 0,Y 447.599,Z 66.888,A -85,B 0,C 180,E1 -8553.629,E2 -8553.629} C_VEL
LIN {X 0,Y 447.58,Z 62.995,A -85,B 0,C 180,E1 -8554.503,E2 -8554.503} C_VEL
LIN {X 0,Y 446.64,Z 56.853,A -85,B 0,C 180,E1 -8555.984,E2 -8555.984} C_VEL
LIN {X 0,Y 446.606,Z 56.855,A -85,B 0,C 180,E1 -8558.142,E2 -8558.142} C_VEL
LIN {X 0,Y 446.523,Z 56.861,A -85,B 0,C 180,E1 -8561.807,E2 -8561.807} C_VEL
LIN {X 0,Y 446.514,Z 56.861,A -85,B 0,C 180,E1 -8565.52,E2 -8565.52} C_VEL
LIN {X 0,Y 446.48,Z 56.865,A -85,B 0,C 180,E1 -8569.185,E2 -8569.185} C_VEL
LIN {X 0,Y 446.424,Z 56.88,A -85,B 0,C 180,E1 -8572.2,E2 -8572.2} C_VEL
LIN {X 0,Y 446.45,Z 56.869,A -85,B 0,C 180,E1 -8575.153,E2 -8575.153} C_VEL
LIN {X 0,Y 446.49,Z 56.869,A -85,B 0,C 180,E1 -8578.179,E2 -8578.179} C_VEL
LIN {X 0,Y 446.424,Z 56.879,A -85,B 0,C 180,E1 -8581.775,E2 -8581.775} C_VEL
LIN {X 0,Y 446.435,Z 56.871,A -85,B 0,C 180,E1 -8584.523,E2 -8584.523} C_VEL
LIN {X 0,Y 446.435,Z 56.873,A -85,B 0,C 180,E1 -8588.082,E2 -8588.082} C_VEL
LIN {X 0,Y 446.431,Z 56.873,A -85,B 0,C 180,E1 -8590.917,E2 -8590.917} C_VEL
LIN {X 0,Y 446.404,Z 56.877,A -85,B 0,C 180,E1 -8593.846,E2 -8593.846} C_VEL
LIN {X 0,Y 446.402,Z 56.875,A -85,B 0,C 180,E1 -8596.403,E2 -8596.403} C_VEL
LIN {X 0,Y 446.431,Z 56.877,A -85,B 0,C 180,E1 -8599.082,E2 -8599.082} C_VEL
LIN {X 0,Y 446.413,Z 56.874,A -85,B 0,C 180,E1 -8602.121,E2 -8602.121} C_VEL
LIN {X 0,Y 446.433,Z 56.873,A -85,B 0,C 180,E1 -8605.477,E2 -8605.477} C_VEL
LIN {X 0,Y 446.42,Z 56.878,A -85,B 0,C 180,E1 -8608.699,E2 -8608.699} C_VEL
LIN {X 0,Y 446.488,Z 56.864,A -85,B 0,C 180,E1 -8611.821,E2 -8611.821} C_VEL
LIN {X 0,Y 446.462,Z 56.873,A -85,B 0,C 180,E1 -8614.848,E2 -8614.848} C_VEL
LIN {X 0,Y 446.451,Z 56.873,A -85,B 0,C 180,E1 -8618.245,E2 -8618.245} C_VEL
LIN {X 0,Y 446.459,Z 56.868,A -85,B 0,C 180,E1 -8621.649,E2 -8621.649} C_VEL
LIN {X 0,Y 446.511,Z 56.867,A -85,B 0,C 180,E1 -8624.48,E2 -8624.48} C_VEL
LIN {X 0,Y 446.52,Z 56.868,A -85,B 0,C 180,E1 -8628.193,E2 -8628.193} C_VEL
LIN {X 0,Y 446.603,Z 56.855,A -85,B 0,C 180,E1 -8631.858,E2 -8631.858} C_VEL
LIN {X 0,Y 446.645,Z 56.846,A -85,B 0,C 180,E1 -8634.582,E2 -8634.582} C_VEL
LIN {X 0,Y 446.665,Z 56.846,A -85,B 0,C 180,E1 -8638.196,E2 -8638.196} C_VEL
LIN {X 0,Y 446.794,Z 56.831,A -85,B 0,C 180,E1 -8640,E2 -8640} C_VEL
LIN {X 0,Y 446.692,Z 56.839,A -85,B 0,C 180,E1 -8642.705,E2 -8642.705} C_VEL
LIN {X 0,Y 446.636,Z 56.846,A -85,B 0,C 180,E1 -8646.324,E2 -8646.324} C_VEL
LIN {X 0,Y 446.535,Z 56.861,A -85,B 0,C 180,E1 -8649.055,E2 -8649.055} C_VEL
LIN {X 0,Y 446.524,Z 56.861,A -85,B 0,C 180,E1 -8652.73,E2 -8652.73} C_VEL
LIN {X 0,Y 446.498,Z 56.863,A -85,B 0,C 180,E1 -8656.227,E2 -8656.227} C_VEL
LIN {X 0,Y 446.47,Z 56.872,A -85,B 0,C 180,E1 -8659.303,E2 -8659.303} C_VEL
LIN {X 0,Y 446.42,Z 56.873,A -85,B 0,C 180,E1 -8662.199,E2 -8662.199} C_VEL
LIN {X 0,Y 446.446,Z 56.874,A -85,B 0,C 180,E1 -8665.153,E2 -8665.153} C_VEL
LIN {X 0,Y 446.486,Z 56.866,A -85,B 0,C 180,E1 -8668.178,E2 -8668.178} C_VEL
LIN {X 0,Y 446.421,Z 56.873,A -85,B 0,C 180,E1 -8671.775,E2 -8671.775} C_VEL
LIN {X 0,Y 446.431,Z 56.878,A -85,B 0,C 180,E1 -8674.523,E2 -8674.523} C_VEL
LIN {X 0,Y 446.415,Z 56.877,A -85,B 0,C 180,E1 -8678.079,E2 -8678.079} C_VEL
LIN {X 0,Y 446.428,Z 56.873,A -85,B 0,C 180,E1 -8680.917,E2 -8680.917} C_VEL
LIN {X 0,Y 446.4,Z 56.878,A -85,B 0,C 180,E1 -8683.846,E2 -8683.846} C_VEL
LIN {X 0,Y 446.398,Z 56.88,A -85,B 0,C 180,E1 -8686.404,E2 -8686.404} C_VEL
LIN {X 0,Y 446.429,Z 56.872,A -85,B 0,C 180,E1 -8689.082,E2 -8689.082} C_VEL
LIN {X 0,Y 446.411,Z 56.879,A -85,B 0,C 180,E1 -8692.121,E2 -8692.121} C_VEL
LIN {X 0,Y 446.431,Z 56.875,A -85,B 0,C 180,E1 -8695.477,E2 -8695.477} C_VEL
LIN {X 0,Y 446.418,Z 56.873,A -85,B 0,C 180,E1 -8698.699,E2 -8698.699} C_VEL
LIN {X 0,Y 446.517,Z 56.868,A -85,B 0,C 180,E1 -8702.334,E2 -8702.334} C_VEL
LIN {X 0,Y 446.571,Z 56.923,A -85,B 0,C 180,E1 -8702.782,E2 -8702.782} C_VEL
LIN {X 0,Y 448.953,Z 70.096,A -85,B 0,C 180,E1 -8705.223,E2 -8705.223} C_VEL
LIN {X 0,Y 448.111,Z 88.408,A -85,B 0,C 180,E1 -8708.373,E2 -8708.373} C_VEL
LIN {X 0,Y 447.275,Z 107.893,A -85,B 0,C 180,E1 -8711.684,E2 -8711.684} C_VEL
LIN {X 0,Y 447.114,Z 111.881,A -85,B 0,C 180,E1 -8712.357,E2 -8712.357} C_VEL
LIN {X 0,Y 450.351,Z 136.353,A -85,B 0,C 180,E1 -8712.866,E2 -8712.866} C_VEL
LIN {X 0,Y 449.563,Z 221.003,A -85,B 0,C 180,E1 -8714.239,E2 -8714.239} C_VEL
LIN {X 0,Y 449.175,Z 233.446,A -85,B 0,C 180,E1 -8714.603,E2 -8714.603} C_VEL
LIN {X 0,Y 448.679,Z 245.799,A -85,B 0,C 180,E1 -8715.138,E2 -8715.138} C_VEL
LIN {X 0,Y 448.145,Z 257.409,A -85,B 0,C 180,E1 -8715.816,E2 -8715.816} C_VEL
LIN {X 0,Y 447.588,Z 268.656,A -85,B 0,C 180,E1 -8716.666,E2 -8716.666} C_VEL
LIN {X 0,Y 446.959,Z 279.949,A -85,B 0,C 180,E1 -8717.744,E2 -8717.744} C_VEL
LIN {X 0,Y 446.502,Z 289.549,A -85,B 0,C 180,E1 -8718.882,E2 -8718.882} C_VEL
LIN {X 0,Y 446.001,Z 298.772,A -85,B 0,C 180,E1 -8720.247,E2 -8720.247} C_VEL
LIN {X 0,Y 445.752,Z 306.205,A -85,B 0,C 180,E1 -8721.614,E2 -8721.614} C_VEL
LIN {X 0,Y 445.509,Z 313.016,A -85,B 0,C 180,E1 -8723.205,E2 -8723.205} C_VEL
LIN {X 0,Y 445.465,Z 317.51,A -85,B 0,C 180,E1 -8724.568,E2 -8724.568} C_VEL
LIN {X 0,Y 445.419,Z 319.875,A -85,B 0,C 180,E1 -8725.475,E2 -8725.475} C_VEL
LIN {X 0,Y 445.452,Z 321.81,A -85,B 0,C 180,E1 -8726.381,E2 -8726.381} C_VEL
LIN {X 0,Y 445.477,Z 323.304,A -85,B 0,C 180,E1 -8727.287,E2 -8727.287} C_VEL
LIN {X 0,Y 445.455,Z 324.347,A -85,B 0,C 180,E1 -8728.191,E2 -8728.191} C_VEL
LIN {X 0,Y 445.441,Z 324.997,A -85,B 0,C 180,E1 -8729.096,E2 -8729.096} C_VEL
LIN {X 0,Y 445.422,Z 325.257,A -85,B 0,C 180,E1 -8730,E2 -8730} C_VEL
LIN {X 0,Y 445.44,Z 325.114,A -85,B 0,C 180,E1 -8730.904,E2 -8730.904} C_VEL
LIN {X 0,Y 445.475,Z 323.574,A -85,B 0,C 180,E1 -8732.712,E2 -8732.712} C_VEL
LIN {X 0,Y 445.433,Z 322.208,A -85,B 0,C 180,E1 -8733.618,E2 -8733.618} C_VEL
LIN {X 0,Y 445.465,Z 319.333,A -85,B 0,C 180,E1 -8734.978,E2 -8734.978} C_VEL
LIN {X 0,Y 445.454,Z 315.428,A -85,B 0,C 180,E1 -8736.34,E2 -8736.34} C_VEL
LIN {X 0,Y 445.669,Z 310.405,A -85,B 0,C 180,E1 -8737.703,E2 -8737.703} C_VEL
LIN {X 0,Y 445.886,Z 304.106,A -85,B 0,C 180,E1 -8739.068,E2 -8739.068} C_VEL
LIN {X 0,Y 446.268,Z 296.252,A -85,B 0,C 180,E1 -8740.434,E2 -8740.434} C_VEL
LIN {X 0,Y 446.925,Z 286.475,A -85,B 0,C 180,E1 -8741.796,E2 -8741.796} C_VEL
LIN {X 0,Y 447.439,Z 276.997,A -85,B 0,C 180,E1 -8742.87,E2 -8742.87} C_VEL
LIN {X 0,Y 448.125,Z 266.408,A -85,B 0,C 180,E1 -8743.837,E2 -8743.837} C_VEL
LIN {X 0,Y 448.833,Z 253.829,A -85,B 0,C 180,E1 -8744.741,E2 -8744.741} C_VEL
LIN {X 0,Y 449.508,Z 241.394,A -85,B 0,C 180,E1 -8745.414,E2 -8745.414} C_VEL
LIN {X 0,Y 450.08,Z 229.055,A -85,B 0,C 180,E1 -8745.887,E2 -8745.887} C_VEL
LIN {X 0,Y 450.455,Z 215.312,A -85,B 0,C 180,E1 -8746.222,E2 -8746.222} C_VEL
LIN {X 0,Y 451.141,Z 135.696,A -85,B 0,C 180,E1 -8747.518,E2 -8747.518} C_VEL
LIN {X 0,Y 448.131,Z 115.393,A -85,B 0,C 180,E1 -8747.995,E2 -8747.995} C_VEL
LIN {X 0,Y 447.428,Z 111.302,A -85,B 0,C 180,E1 -8748.115,E2 -8748.115} C_VEL
LIN {X 0,Y 448.247,Z 95.237,A -85,B 0,C 180,E1 -8750.897,E2 -8750.897} C_VEL
LIN {X 0,Y 449.343,Z 76.248,A -85,B 0,C 180,E1 -8754.238,E2 -8754.238} C_VEL
LIN {X 0,Y 449.445,Z 70.813,A -85,B 0,C 180,E1 -8755.221,E2 -8755.221} C_VEL
LIN {X 0,Y 447.238,Z 59.957,A -85,B 0,C 180,E1 -8757.364,E2 -8757.364} C_VEL
LIN {X 0,Y 446.493,Z 56.871,A -85,B 0,C 180,E1 -8758.006,E2 -8758.006} C_VEL
LIN {X 0,Y 446.416,Z 56.88,A -85,B 0,C 180,E1 -8761.3,E2 -8761.3} C_VEL
LIN {X 0,Y 446.429,Z 56.874,A -85,B 0,C 180,E1 -8764.522,E2 -8764.522} C_VEL
LIN {X 0,Y 446.43,Z 56.878,A -85,B 0,C 180,E1 -8768.081,E2 -8768.081} C_VEL
LIN {X 0,Y 446.425,Z 56.874,A -85,B 0,C 180,E1 -8770.917,E2 -8770.917} C_VEL
LIN {X 0,Y 446.399,Z 56.879,A -85,B 0,C 180,E1 -8773.846,E2 -8773.846} C_VEL
LIN {X 0,Y 446.396,Z 56.874,A -85,B 0,C 180,E1 -8776.403,E2 -8776.403} C_VEL
LIN {X 0,Y 446.466,Z 56.871,A -85,B 0,C 180,E1 -8779.805,E2 -8779.805} C_VEL
LIN {X 0,Y 446.431,Z 56.87,A -85,B 0,C 180,E1 -8782.123,E2 -8782.123} C_VEL
LIN {X 0,Y 446.429,Z 56.874,A -85,B 0,C 180,E1 -8785.477,E2 -8785.477} C_VEL
LIN {X 0,Y 446.414,Z 56.878,A -85,B 0,C 180,E1 -8788.7,E2 -8788.7} C_VEL
LIN {X 0,Y 446.482,Z 56.866,A -85,B 0,C 180,E1 -8791.821,E2 -8791.821} C_VEL
LIN {X 0,Y 446.456,Z 56.875,A -85,B 0,C 180,E1 -8794.848,E2 -8794.848} C_VEL
LIN {X 0,Y 446.446,Z 56.867,A -85,B 0,C 180,E1 -8798.245,E2 -8798.245} C_VEL
LIN {X 0,Y 446.455,Z 56.866,A -85,B 0,C 180,E1 -8801.649,E2 -8801.649} C_VEL
LIN {X 0,Y 446.505,Z 56.869,A -85,B 0,C 180,E1 -8804.48,E2 -8804.48} C_VEL
LIN {X 0,Y 446.515,Z 56.862,A -85,B 0,C 180,E1 -8808.193,E2 -8808.193} C_VEL
LIN {X 0,Y 446.598,Z 56.852,A -85,B 0,C 180,E1 -8811.858,E2 -8811.858} C_VEL
LIN {X 0,Y 446.641,Z 56.848,A -85,B 0,C 180,E1 -8814.583,E2 -8814.583} C_VEL
LIN {X 0,Y 446.661,Z 56.844,A -85,B 0,C 180,E1 -8818.197,E2 -8818.197} C_VEL
LIN {X 0,Y 446.79,Z 56.832,A -85,B 0,C 180,E1 -8820,E2 -8820} C_VEL
LIN {X 0,Y 446.688,Z 56.834,A -85,B 0,C 180,E1 -8822.706,E2 -8822.706} C_VEL
LIN {X 0,Y 446.632,Z 56.847,A -85,B 0,C 180,E1 -8826.324,E2 -8826.324} C_VEL
LIN {X 0,Y 446.531,Z 56.858,A -85,B 0,C 180,E1 -8829.056,E2 -8829.056} C_VEL
LIN {X 0,Y 446.519,Z 56.861,A -85,B 0,C 180,E1 -8832.73,E2 -8832.73} C_VEL
LIN {X 0,Y 446.494,Z 56.864,A -85,B 0,C 180,E1 -8836.228,E2 -8836.228} C_VEL
LIN {X 0,Y 446.466,Z 56.871,A -85,B 0,C 180,E1 -8839.304,E2 -8839.304} C_VEL
LIN {X 0,Y 446.416,Z 56.87,A -85,B 0,C 180,E1 -8842.2,E2 -8842.2} C_VEL
LIN {X 0,Y 446.441,Z 56.869,A -85,B 0,C 180,E1 -8845.154,E2 -8845.154} C_VEL
LIN {X 0,Y 446.448,Z 56.874,A -85,B 0,C 180,E1 -8848.182,E2 -8848.182} C_VEL
LIN {X 0,Y 446.414,Z 56.875,A -85,B 0,C 180,E1 -8851.301,E2 -8851.301} C_VEL
LIN {X 0,Y 446.421,Z 56.876,A -85,B 0,C 180,E1 -8854.524,E2 -8854.524} C_VEL
LIN {X 0,Y 446.409,Z 56.88,A -85,B 0,C 180,E1 -8858.079,E2 -8858.079} C_VEL
LIN {X 0,Y 446.406,Z 56.872,A -85,B 0,C 180,E1 -8861.394,E2 -8861.394} C_VEL
LIN {X 0,Y 446.449,Z 56.87,A -85,B 0,C 180,E1 -8865.105,E2 -8865.105} C_VEL
LIN {X 0,Y 446.407,Z 56.877,A -85,B 0,C 180,E1 -8868.607,E2 -8868.607} C_VEL
LIN {X 0,Y 446.403,Z 56.881,A -85,B 0,C 180,E1 -8871.924,E2 -8871.924} C_VEL
LIN {X 0,Y 446.491,Z 57.072,A -85,B 0,C 180,E1 -8875.483,E2 -8875.483} C_VEL
LIN {X 0,Y 448.036,Z 65.301,A -85,B 0,C 180,E1 -8877.504,E2 -8877.504} C_VEL
LIN {X 0,Y 448.128,Z 67.344,A -85,B 0,C 180,E1 -8877.981,E2 -8877.981} C_VEL
LIN {X 0,Y 451.69,Z 82.582,A -85,B 0,C 180,E1 -8878.418,E2 -8878.418} C_VEL
LIN {X 0,Y 450.728,Z 173.485,A -85,B 0,C 180,E1 -8879.908,E2 -8879.908} C_VEL
LIN {X 0,Y 450.436,Z 186.775,A -85,B 0,C 180,E1 -8880.306,E2 -8880.306} C_VEL
LIN {X 0,Y 450.064,Z 199.476,A -85,B 0,C 180,E1 -8880.876,E2 -8880.876} C_VEL
LIN {X 0,Y 449.55,Z 210.284,A -85,B 0,C 180,E1 -8881.523,E2 -8881.523} C_VEL
LIN {X 0,Y 448.887,Z 221.308,A -85,B 0,C 180,E1 -8882.366,E2 -8882.366} C_VEL
LIN {X 0,Y 448.282,Z 232.377,A -85,B 0,C 180,E1 -8883.443,E2 -8883.443} C_VEL
LIN {X 0,Y 447.632,Z 242.491,A -85,B 0,C 180,E1 -8884.67,E2 -8884.67} C_VEL
LIN {X 0,Y 447.119,Z 250.505,A -85,B 0,C 180,E1 -8885.879,E2 -8885.879} C_VEL
LIN {X 0,Y 446.609,Z 257.774,A -85,B 0,C 180,E1 -8887.223,E2 -8887.223} C_VEL
LIN {X 0,Y 445.785,Z 260.845,A -85,B 0,C 180,E1 -8887.865,E2 -8887.865} C_VEL
LIN {X 0,Y 442.672,Z 265.435,A -85,B 0,C 180,E1 -8888.927,E2 -8888.927} C_VEL
LIN {X 0,Y 439.566,Z 269.376,A -85,B 0,C 180,E1 -8890.043,E2 -8890.043} C_VEL
LIN {X 0,Y 438.763,Z 271.312,A -85,B 0,C 180,E1 -8890.763,E2 -8890.763} C_VEL
LIN {X 0,Y 438.491,Z 274.456,A -85,B 0,C 180,E1 -8892.271,E2 -8892.271} C_VEL
LIN {X 0,Y 438.429,Z 275.822,A -85,B 0,C 180,E1 -8893.23,E2 -8893.23} C_VEL
LIN {X 0,Y 438.367,Z 276.773,A -85,B 0,C 180,E1 -8894.184,E2 -8894.184} C_VEL
LIN {X 0,Y 438.336,Z 277.308,A -85,B 0,C 180,E1 -8895.136,E2 -8895.136} C_VEL
LIN {X 0,Y 438.326,Z 277.386,A -85,B 0,C 180,E1 -8896.084,E2 -8896.084} C_VEL
LIN {X 0,Y 438.426,Z 276.344,A -85,B 0,C 180,E1 -8897.972,E2 -8897.972} C_VEL
LIN {X 0,Y 438.448,Z 275.201,A -85,B 0,C 180,E1 -8898.91,E2 -8898.91} C_VEL
LIN {X 0,Y 438.533,Z 272.693,A -85,B 0,C 180,E1 -8900.313,E2 -8900.313} C_VEL
LIN {X 0,Y 438.724,Z 269.168,A -85,B 0,C 180,E1 -8901.711,E2 -8901.711} C_VEL
LIN {X 0,Y 438.921,Z 264.566,A -85,B 0,C 180,E1 -8903.098,E2 -8903.098} C_VEL
LIN {X 0,Y 439.275,Z 257.568,A -85,B 0,C 180,E1 -8904.722,E2 -8904.722} C_VEL
LIN {X 0,Y 439.696,Z 250.031,A -85,B 0,C 180,E1 -8906.105,E2 -8906.105} C_VEL
LIN {X 0,Y 440.188,Z 242.317,A -85,B 0,C 180,E1 -8907.255,E2 -8907.255} C_VEL
LIN {X 0,Y 440.828,Z 231.845,A -85,B 0,C 180,E1 -8908.516,E2 -8908.516} C_VEL
LIN {X 0,Y 441.41,Z 221.206,A -85,B 0,C 180,E1 -8909.544,E2 -8909.544} C_VEL
LIN {X 0,Y 441.929,Z 210.901,A -85,B 0,C 180,E1 -8910.342,E2 -8910.342} C_VEL
LIN {X 0,Y 442.359,Z 198.608,A -85,B 0,C 180,E1 -8911.081,E2 -8911.081} C_VEL
LIN {X 0,Y 442.661,Z 185.723,A -85,B 0,C 180,E1 -8911.649,E2 -8911.649} C_VEL
LIN {X 0,Y 442.992,Z 172.936,A -85,B 0,C 180,E1 -8912.018,E2 -8912.018} C_VEL
LIN {X 0,Y 443.767,Z 82.988,A -85,B 0,C 180,E1 -8913.496,E2 -8913.496} C_VEL
LIN {X 0,Y 440.63,Z 67.185,A -85,B 0,C 180,E1 -8913.887,E2 -8913.887} C_VEL
LIN {X 0,Y 440.301,Z 62.193,A -85,B 0,C 180,E1 -8915.037,E2 -8915.037} C_VEL
LIN {X 0,Y 439.605,Z 57.729,A -85,B 0,C 180,E1 -8916.138,E2 -8916.138} C_VEL
LIN {X 0,Y 439.554,Z 57.735,A -85,B 0,C 180,E1 -8918.274,E2 -8918.274} C_VEL
LIN {X 0,Y 439.489,Z 57.738,A -85,B 0,C 180,E1 -8921.999,E2 -8921.999} C_VEL
LIN {X 0,Y 439.468,Z 57.74,A -85,B 0,C 180,E1 -8925.776,E2 -8925.776} C_VEL
LIN {X 0,Y 439.446,Z 57.742,A -85,B 0,C 180,E1 -8929.337,E2 -8929.337} C_VEL
LIN {X 0,Y 439.37,Z 57.754,A -85,B 0,C 180,E1 -8932.575,E2 -8932.575} C_VEL
LIN {X 0,Y 439.403,Z 57.749,A -85,B 0,C 180,E1 -8935.585,E2 -8935.585} C_VEL
LIN {X 0,Y 439.422,Z 57.745,A -85,B 0,C 180,E1 -8938.673,E2 -8938.673} C_VEL
LIN {X 0,Y 439.375,Z 57.755,A -85,B 0,C 180,E1 -8942.03,E2 -8942.03} C_VEL
LIN {X 0,Y 439.401,Z 57.75,A -85,B 0,C 180,E1 -8945.341,E2 -8945.341} C_VEL
LIN {X 0,Y 439.395,Z 57.748,A -85,B 0,C 180,E1 -8948.594,E2 -8948.594} C_VEL
LIN {X 0,Y 439.393,Z 57.753,A -85,B 0,C 180,E1 -8951.257,E2 -8951.257} C_VEL
LIN {X 0,Y 439.404,Z 57.748,A -85,B 0,C 180,E1 -8954.729,E2 -8954.729} C_VEL
LIN {X 0,Y 439.4,Z 57.749,A -85,B 0,C 180,E1 -8957.795,E2 -8957.795} C_VEL
LIN {X 0,Y 439.43,Z 57.744,A -85,B 0,C 180,E1 -8960.227,E2 -8960.227} C_VEL
LIN {X 0,Y 439.377,Z 57.751,A -85,B 0,C 180,E1 -8963.713,E2 -8963.713} C_VEL
LIN {X 0,Y 439.376,Z 57.756,A -85,B 0,C 180,E1 -8967.054,E2 -8967.054} C_VEL
LIN {X 0,Y 439.386,Z 57.751,A -85,B 0,C 180,E1 -8970.274,E2 -8970.274} C_VEL
LIN {X 0,Y 439.432,Z 57.744,A -85,B 0,C 180,E1 -8973.396,E2 -8973.396} C_VEL
LIN {X 0,Y 439.391,Z 57.754,A -85,B 0,C 180,E1 -8976.429,E2 -8976.429} C_VEL
LIN {X 0,Y 439.391,Z 57.749,A -85,B 0,C 180,E1 -8979.397,E2 -8979.397} C_VEL
LIN {X 0,Y 439.434,Z 57.749,A -85,B 0,C 180,E1 -8982.309,E2 -8982.309} C_VEL
LIN {X 0,Y 439.45,Z 57.741,A -85,B 0,C 180,E1 -8985.174,E2 -8985.174} C_VEL
LIN {X 0,Y 439.486,Z 57.741,A -85,B 0,C 180,E1 -8988.001,E2 -8988.001} C_VEL
LIN {X 0,Y 439.55,Z 57.732,A -85,B 0,C 180,E1 -8991.726,E2 -8991.726} C_VEL
LIN {X 0,Y 439.62,Z 57.722,A -85,B 0,C 180,E1 -8994.496,E2 -8994.496} C_VEL
LIN {X 0,Y 439.635,Z 57.722,A -85,B 0,C 180,E1 -8998.168,E2 -8998.168} C_VEL
LIN {X 0,Y 439.764,Z 57.707,A -85,B 0,C 180,E1 -9000,E2 -9000} C_VEL
LIN {X 0,Y 439.641,Z 57.717,A -85,B 0,C 180,E1 -9002.749,E2 -9002.749} C_VEL
LIN {X 0,Y 439.607,Z 57.722,A -85,B 0,C 180,E1 -9006.425,E2 -9006.425} C_VEL
LIN {X 0,Y 439.498,Z 57.739,A -85,B 0,C 180,E1 -9009.201,E2 -9009.201} C_VEL
LIN {X 0,Y 439.468,Z 57.742,A -85,B 0,C 180,E1 -9012.937,E2 -9012.937} C_VEL
LIN {X 0,Y 439.448,Z 57.741,A -85,B 0,C 180,E1 -9016.348,E2 -9016.348} C_VEL
LIN {X 0,Y 439.404,Z 57.749,A -85,B 0,C 180,E1 -9019.626,E2 -9019.626} C_VEL
LIN {X 0,Y 439.366,Z 57.754,A -85,B 0,C 180,E1 -9022.575,E2 -9022.575} C_VEL
LIN {X 0,Y 439.391,Z 57.749,A -85,B 0,C 180,E1 -9025.586,E2 -9025.586} C_VEL
LIN {X 0,Y 439.419,Z 57.751,A -85,B 0,C 180,E1 -9028.673,E2 -9028.673} C_VEL
LIN {X 0,Y 439.372,Z 57.752,A -85,B 0,C 180,E1 -9032.03,E2 -9032.03} C_VEL
LIN {X 0,Y 439.396,Z 57.748,A -85,B 0,C 180,E1 -9035.34,E2 -9035.34} C_VEL
LIN {X 0,Y 439.377,Z 57.756,A -85,B 0,C 180,E1 -9038.596,E2 -9038.596} C_VEL
LIN {X 0,Y 439.39,Z 57.749,A -85,B 0,C 180,E1 -9041.257,E2 -9041.257} C_VEL
LIN {X 0,Y 439.401,Z 57.749,A -85,B 0,C 180,E1 -9044.729,E2 -9044.729} C_VEL
LIN {X 0,Y 439.398,Z 57.751,A -85,B 0,C 180,E1 -9047.796,E2 -9047.796} C_VEL
LIN {X 0,Y 439.428,Z 57.749,A -85,B 0,C 180,E1 -9050.227,E2 -9050.227} C_VEL
LIN {X 0,Y 439.376,Z 57.755,A -85,B 0,C 180,E1 -9053.713,E2 -9053.713} C_VEL
LIN {X 0,Y 439.374,Z 57.751,A -85,B 0,C 180,E1 -9057.054,E2 -9057.054} C_VEL
LIN {X 0,Y 439.384,Z 57.757,A -85,B 0,C 180,E1 -9060.274,E2 -9060.274} C_VEL
LIN {X 0,Y 439.511,Z 57.843,A -85,B 0,C 180,E1 -9062.598,E2 -9062.598} C_VEL
LIN {X 0,Y 441.945,Z 70.655,A -85,B 0,C 180,E1 -9065.018,E2 -9065.018} C_VEL
LIN {X 0,Y 441.257,Z 87.799,A -85,B 0,C 180,E1 -9068.019,E2 -9068.019} C_VEL
LIN {X 0,Y 440.243,Z 108.674,A -85,B 0,C 180,E1 -9071.622,E2 -9071.622} C_VEL
LIN {X 0,Y 440.153,Z 111.792,A -85,B 0,C 180,E1 -9072.114,E2 -9072.114} C_VEL
LIN {X 0,Y 443.501,Z 137.15,A -85,B 0,C 180,E1 -9072.651,E2 -9072.651} C_VEL
LIN {X 0,Y 442.665,Z 220.267,A -85,B 0,C 180,E1 -9074.016,E2 -9074.016} C_VEL
LIN {X 0,Y 442.254,Z 233.603,A -85,B 0,C 180,E1 -9074.415,E2 -9074.415} C_VEL
LIN {X 0,Y 441.741,Z 245.829,A -85,B 0,C 180,E1 -9074.958,E2 -9074.958} C_VEL
LIN {X 0,Y 441.126,Z 258.161,A -85,B 0,C 180,E1 -9075.703,E2 -9075.703} C_VEL
LIN {X 0,Y 440.538,Z 269.588,A -85,B 0,C 180,E1 -9076.603,E2 -9076.603} C_VEL
LIN {X 0,Y 439.914,Z 280.328,A -85,B 0,C 180,E1 -9077.662,E2 -9077.662} C_VEL
LIN {X 0,Y 439.478,Z 288.914,A -85,B 0,C 180,E1 -9078.702,E2 -9078.702} C_VEL
LIN {X 0,Y 438.947,Z 298.2,A -85,B 0,C 180,E1 -9080.089,E2 -9080.089} C_VEL
LIN {X 0,Y 438.671,Z 305.67,A -85,B 0,C 180,E1 -9081.477,E2 -9081.477} C_VEL
LIN {X 0,Y 438.442,Z 312.525,A -85,B 0,C 180,E1 -9083.095,E2 -9083.095} C_VEL
LIN {X 0,Y 438.355,Z 317.041,A -85,B 0,C 180,E1 -9084.48,E2 -9084.48} C_VEL
LIN {X 0,Y 438.346,Z 319.422,A -85,B 0,C 180,E1 -9085.402,E2 -9085.402} C_VEL
LIN {X 0,Y 438.352,Z 321.367,A -85,B 0,C 180,E1 -9086.323,E2 -9086.323} C_VEL
LIN {X 0,Y 438.403,Z 322.882,A -85,B 0,C 180,E1 -9087.243,E2 -9087.243} C_VEL
LIN {X 0,Y 438.379,Z 324.598,A -85,B 0,C 180,E1 -9089.081,E2 -9089.081} C_VEL
LIN {X 0,Y 438.359,Z 324.868,A -85,B 0,C 180,E1 -9090,E2 -9090} C_VEL
LIN {X 0,Y 438.348,Z 324.741,A -85,B 0,C 180,E1 -9090.918,E2 -9090.918} C_VEL
LIN {X 0,Y 438.4,Z 323.224,A -85,B 0,C 180,E1 -9092.756,E2 -9092.756} C_VEL
LIN {X 0,Y 438.332,Z 321.867,A -85,B 0,C 180,E1 -9093.677,E2 -9093.677} C_VEL
LIN {X 0,Y 438.367,Z 319.013,A -85,B 0,C 180,E1 -9095.058,E2 -9095.058} C_VEL
LIN {X 0,Y 438.368,Z 315.133,A -85,B 0,C 180,E1 -9096.443,E2 -9096.443} C_VEL
LIN {X 0,Y 438.587,Z 310.14,A -85,B 0,C 180,E1 -9097.828,E2 -9097.828} C_VEL
LIN {X 0,Y 438.834,Z 303.877,A -85,B 0,C 180,E1 -9099.215,E2 -9099.215} C_VEL
LIN {X 0,Y 439.269,Z 296.088,A -85,B 0,C 180,E1 -9100.602,E2 -9100.602} C_VEL
LIN {X 0,Y 439.963,Z 286.365,A -85,B 0,C 180,E1 -9101.985,E2 -9101.985} C_VEL
LIN {X 0,Y 440.563,Z 276.15,A -85,B 0,C 180,E1 -9103.16,E2 -9103.16} C_VEL
LIN {X 0,Y 441.318,Z 265.04,A -85,B 0,C 180,E1 -9104.172,E2 -9104.172} C_VEL
LIN {X 0,Y 441.973,Z 253.993,A -85,B 0,C 180,E1 -9104.975,E2 -9104.975} C_VEL
LIN {X 0,Y 442.697,Z 241.762,A -85,B 0,C 180,E1 -9105.657,E2 -9105.657} C_VEL
LIN {X 0,Y 443.334,Z 228.902,A -85,B 0,C 180,E1 -9106.165,E2 -9106.165} C_VEL
LIN {X 0,Y 443.71,Z 215.317,A -85,B 0,C 180,E1 -9106.506,E2 -9106.506} C_VEL
LIN {X 0,Y 444.435,Z 136.359,A -85,B 0,C 180,E1 -9107.812,E2 -9107.812} C_VEL
LIN {X 0,Y 441.515,Z 116.569,A -85,B 0,C 180,E1 -9108.288,E2 -9108.288} C_VEL
LIN {X 0,Y 440.554,Z 110.932,A -85,B 0,C 180,E1 -9108.444,E2 -9108.444} C_VEL
LIN {X 0,Y 441.529,Z 92.405,A -85,B 0,C 180,E1 -9111.72,E2 -9111.72} C_VEL
LIN {X 0,Y 442.649,Z 74.079,A -85,B 0,C 180,E1 -9115.013,E2 -9115.013} C_VEL
LIN {X 0,Y 441.987,Z 69.368,A -85,B 0,C 180,E1 -9115.93,E2 -9115.93} C_VEL
LIN {X 0,Y 439.443,Z 57.751,A -85,B 0,C 180,E1 -9118.311,E2 -9118.311} C_VEL
LIN {X 0,Y 439.372,Z 57.761,A -85,B 0,C 180,E1 -9121.86,E2 -9121.86} C_VEL
LIN {X 0,Y 439.4,Z 57.747,A -85,B 0,C 180,E1 -9125.155,E2 -9125.155} C_VEL
LIN {X 0,Y 439.389,Z 57.751,A -85,B 0,C 180,E1 -9128.594,E2 -9128.594} C_VEL
LIN {X 0,Y 439.387,Z 57.753,A -85,B 0,C 180,E1 -9131.256,E2 -9131.256} C_VEL
LIN {X 0,Y 439.398,Z 57.746,A -85,B 0,C 180,E1 -9134.729,E2 -9134.729} C_VEL
LIN {X 0,Y 439.395,Z 57.753,A -85,B 0,C 180,E1 -9137.796,E2 -9137.796} C_VEL
LIN {X 0,Y 439.449,Z 57.742,A -85,B 0,C 180,E1 -9140.23,E2 -9140.23} C_VEL
LIN {X 0,Y 439.375,Z 57.754,A -85,B 0,C 180,E1 -9143.713,E2 -9143.713} C_VEL
LIN {X 0,Y 439.371,Z 57.756,A -85,B 0,C 180,E1 -9147.054,E2 -9147.054} C_VEL
LIN {X 0,Y 439.38,Z 57.75,A -85,B 0,C 180,E1 -9150.274,E2 -9150.274} C_VEL
LIN {X 0,Y 439.427,Z 57.743,A -85,B 0,C 180,E1 -9153.396,E2 -9153.396} C_VEL
LIN {X 0,Y 439.385,Z 57.754,A -85,B 0,C 180,E1 -9156.43,E2 -9156.43} C_VEL
LIN {X 0,Y 439.386,Z 57.75,A -85,B 0,C 180,E1 -9159.397,E2 -9159.397} C_VEL
LIN {X 0,Y 439.429,Z 57.743,A -85,B 0,C 180,E1 -9162.31,E2 -9162.31} C_VEL
LIN {X 0,Y 439.445,Z 57.743,A -85,B 0,C 180,E1 -9165.174,E2 -9165.174} C_VEL
LIN {X 0,Y 439.481,Z 57.735,A -85,B 0,C 180,E1 -9168.001,E2 -9168.001} C_VEL
LIN {X 0,Y 439.546,Z 57.731,A -85,B 0,C 180,E1 -9171.726,E2 -9171.726} C_VEL
LIN {X 0,Y 439.616,Z 57.723,A -85,B 0,C 180,E1 -9174.496,E2 -9174.496} C_VEL
LIN {X 0,Y 439.631,Z 57.72,A -85,B 0,C 180,E1 -9178.168,E2 -9178.168} C_VEL
LIN {X 0,Y 439.759,Z 57.708,A -85,B 0,C 180,E1 -9180,E2 -9180} C_VEL
LIN {X 0,Y 439.637,Z 57.712,A -85,B 0,C 180,E1 -9182.749,E2 -9182.749} C_VEL
LIN {X 0,Y 439.602,Z 57.722,A -85,B 0,C 180,E1 -9186.426,E2 -9186.426} C_VEL
LIN {X 0,Y 439.494,Z 57.736,A -85,B 0,C 180,E1 -9189.202,E2 -9189.202} C_VEL
LIN {X 0,Y 439.463,Z 57.739,A -85,B 0,C 180,E1 -9192.938,E2 -9192.938} C_VEL
LIN {X 0,Y 439.444,Z 57.743,A -85,B 0,C 180,E1 -9196.349,E2 -9196.349} C_VEL
LIN {X 0,Y 439.4,Z 57.749,A -85,B 0,C 180,E1 -9199.627,E2 -9199.627} C_VEL
LIN {X 0,Y 439.362,Z 57.752,A -85,B 0,C 180,E1 -9202.576,E2 -9202.576} C_VEL
LIN {X 0,Y 439.379,Z 57.747,A -85,B 0,C 180,E1 -9205.587,E2 -9205.587} C_VEL
LIN {X 0,Y 439.398,Z 57.75,A -85,B 0,C 180,E1 -9208.675,E2 -9208.675} C_VEL
LIN {X 0,Y 439.368,Z 57.756,A -85,B 0,C 180,E1 -9212.031,E2 -9212.031} C_VEL
LIN {X 0,Y 439.39,Z 57.747,A -85,B 0,C 180,E1 -9215.34,E2 -9215.34} C_VEL
LIN {X 0,Y 439.361,Z 57.758,A -85,B 0,C 180,E1 -9218.598,E2 -9218.598} C_VEL
LIN {X 0,Y 439.367,Z 57.748,A -85,B 0,C 180,E1 -9221.254,E2 -9221.254} C_VEL
LIN {X 0,Y 439.397,Z 57.748,A -85,B 0,C 180,E1 -9224.73,E2 -9224.73} C_VEL
LIN {X 0,Y 439.358,Z 57.761,A -85,B 0,C 180,E1 -9227.792,E2 -9227.792} C_VEL
LIN {X 0,Y 439.358,Z 57.759,A -85,B 0,C 180,E1 -9231.403,E2 -9231.403} C_VEL
LIN {X 0,Y 439.396,Z 57.756,A -85,B 0,C 180,E1 -9234.844,E2 -9234.844} C_VEL
LIN {X 0,Y 439.427,Z 57.897,A -85,B 0,C 180,E1 -9235.197,E2 -9235.197} C_VEL
LIN {X 0,Y 441.017,Z 65.838,A -85,B 0,C 180,E1 -9237.193,E2 -9237.193} C_VEL
LIN {X 0,Y 441.19,Z 67.661,A -85,B 0,C 180,E1 -9237.632,E2 -9237.632} C_VEL
LIN {X 0,Y 445.084,Z 83.78,A -85,B 0,C 180,E1 -9238.12,E2 -9238.12} C_VEL
LIN {X 0,Y 444.019,Z 174.49,A -85,B 0,C 180,E1 -9239.635,E2 -9239.635} C_VEL
LIN {X 0,Y 443.706,Z 187.953,A -85,B 0,C 180,E1 -9240.054,E2 -9240.054} C_VEL
LIN {X 0,Y 443.309,Z 200.649,A -85,B 0,C 180,E1 -9240.644,E2 -9240.644} C_VEL
LIN {X 0,Y 442.739,Z 211.666,A -85,B 0,C 180,E1 -9241.329,E2 -9241.329} C_VEL
LIN {X 0,Y 442.009,Z 223.567,A -85,B 0,C 180,E1 -9242.285,E2 -9242.285} C_VEL
LIN {X 0,Y 441.342,Z 234.064,A -85,B 0,C 180,E1 -9243.349,E2 -9243.349} C_VEL
LIN {X 0,Y 440.707,Z 243.186,A -85,B 0,C 180,E1 -9244.497,E2 -9244.497} C_VEL
LIN {X 0,Y 440.127,Z 251.563,A -85,B 0,C 180,E1 -9245.795,E2 -9245.795} C_VEL
LIN {X 0,Y 439.589,Z 258.848,A -85,B 0,C 180,E1 -9247.189,E2 -9247.189} C_VEL
LIN {X 0,Y 439.22,Z 263.993,A -85,B 0,C 180,E1 -9248.407,E2 -9248.407} C_VEL
LIN {X 0,Y 438.955,Z 268.912,A -85,B 0,C 180,E1 -9249.866,E2 -9249.866} C_VEL
LIN {X 0,Y 438.763,Z 271.312,A -85,B 0,C 180,E1 -9250.763,E2 -9250.763} C_VEL
LIN {X 0,Y 437.971,Z 273.059,A -85,B 0,C 180,E1 -9251.493,E2 -9251.493} C_VEL
LIN {X 0,Y 434.932,Z 275.372,A -85,B 0,C 180,E1 -9252.694,E2 -9252.694} C_VEL
LIN {X 0,Y 432.418,Z 276.725,A -85,B 0,C 180,E1 -9253.678,E2 -9253.678} C_VEL
LIN {X 0,Y 431.345,Z 277.385,A -85,B 0,C 180,E1 -9254.447,E2 -9254.447} C_VEL
LIN {X 0,Y 431.258,Z 277.498,A -85,B 0,C 180,E1 -9254.708,E2 -9254.708} C_VEL
LIN {X 0,Y 431.232,Z 277.806,A -85,B 0,C 180,E1 -9255.85,E2 -9255.85} C_VEL
LIN {X 0,Y 431.249,Z 277.551,A -85,B 0,C 180,E1 -9256.812,E2 -9256.812} C_VEL
LIN {X 0,Y 431.324,Z 276.817,A -85,B 0,C 180,E1 -9257.864,E2 -9257.864} C_VEL
LIN {X 0,Y 431.347,Z 275.854,A -85,B 0,C 180,E1 -9258.725,E2 -9258.725} C_VEL
LIN {X 0,Y 431.382,Z 274.372,A -85,B 0,C 180,E1 -9259.677,E2 -9259.677} C_VEL
LIN {X 0,Y 431.558,Z 271.329,A -85,B 0,C 180,E1 -9261.1,E2 -9261.1} C_VEL
LIN {X 0,Y 431.781,Z 267.23,A -85,B 0,C 180,E1 -9262.518,E2 -9262.518} C_VEL
LIN {X 0,Y 432.025,Z 260.973,A -85,B 0,C 180,E1 -9264.165,E2 -9264.165} C_VEL
LIN {X 0,Y 432.46,Z 254.152,A -85,B 0,C 180,E1 -9265.573,E2 -9265.573} C_VEL
LIN {X 0,Y 432.885,Z 247.202,A -85,B 0,C 180,E1 -9266.743,E2 -9266.743} C_VEL
LIN {X 0,Y 433.414,Z 238.837,A -85,B 0,C 180,E1 -9267.909,E2 -9267.909} C_VEL
LIN {X 0,Y 434.061,Z 228.509,A -85,B 0,C 180,E1 -9269.073,E2 -9269.073} C_VEL
LIN {X 0,Y 434.711,Z 216.89,A -85,B 0,C 180,E1 -9270.116,E2 -9270.116} C_VEL
LIN {X 0,Y 435.253,Z 205.339,A -85,B 0,C 180,E1 -9270.926,E2 -9270.926} C_VEL
LIN {X 0,Y 435.658,Z 193.395,A -85,B 0,C 180,E1 -9271.56,E2 -9271.56} C_VEL
LIN {X 0,Y 435.962,Z 181.332,A -85,B 0,C 180,E1 -9272.022,E2 -9272.022} C_VEL
LIN {X 0,Y 436.153,Z 168.155,A -85,B 0,C 180,E1 -9272.338,E2 -9272.338} C_VEL
LIN {X 0,Y 436.865,Z 83.708,A -85,B 0,C 180,E1 -9273.734,E2 -9273.734} C_VEL
LIN {X 0,Y 433.691,Z 67.476,A -85,B 0,C 180,E1 -9274.153,E2 -9274.153} C_VEL
LIN {X 0,Y 433.013,Z 61.377,A -85,B 0,C 180,E1 -9275.589,E2 -9275.589} C_VEL
LIN {X 0,Y 432.58,Z 58.605,A -85,B 0,C 180,E1 -9276.296,E2 -9276.296} C_VEL
LIN {X 0,Y 432.498,Z 58.614,A -85,B 0,C 180,E1 -9278.41,E2 -9278.41} C_VEL
LIN {X 0,Y 432.465,Z 58.615,A -85,B 0,C 180,E1 -9282.197,E2 -9282.197} C_VEL
LIN {X 0,Y 432.436,Z 58.618,A -85,B 0,C 180,E1 -9286.039,E2 -9286.039} C_VEL
LIN {X 0,Y 432.392,Z 58.621,A -85,B 0,C 180,E1 -9289.485,E2 -9289.485} C_VEL
LIN {X 0,Y 432.323,Z 58.629,A -85,B 0,C 180,E1 -9292.964,E2 -9292.964} C_VEL
LIN {X 0,Y 432.367,Z 58.631,A -85,B 0,C 180,E1 -9296.033,E2 -9296.033} C_VEL
LIN {X 0,Y 432.348,Z 58.626,A -85,B 0,C 180,E1 -9299.187,E2 -9299.187} C_VEL
LIN {X 0,Y 432.328,Z 58.629,A -85,B 0,C 180,E1 -9302.443,E2 -9302.443} C_VEL
LIN {X 0,Y 432.35,Z 58.632,A -85,B 0,C 180,E1 -9305.632,E2 -9305.632} C_VEL
LIN {X 0,Y 432.357,Z 58.625,A -85,B 0,C 180,E1 -9308.716,E2 -9308.716} C_VEL
LIN {X 0,Y 432.338,Z 58.631,A -85,B 0,C 180,E1 -9311.797,E2 -9311.797} C_VEL
LIN {X 0,Y 432.337,Z 58.627,A -85,B 0,C 180,E1 -9314.347,E2 -9314.347} C_VEL
LIN {X 0,Y 432.324,Z 58.633,A -85,B 0,C 180,E1 -9317.016,E2 -9317.016} C_VEL
LIN {X 0,Y 432.337,Z 58.628,A -85,B 0,C 180,E1 -9319.821,E2 -9319.821} C_VEL
LIN {X 0,Y 432.31,Z 58.637,A -85,B 0,C 180,E1 -9323.022,E2 -9323.022} C_VEL
LIN {X 0,Y 432.363,Z 58.624,A -85,B 0,C 180,E1 -9325.996,E2 -9325.996} C_VEL
LIN {X 0,Y 432.351,Z 58.627,A -85,B 0,C 180,E1 -9329.489,E2 -9329.489} C_VEL
LIN {X 0,Y 432.394,Z 58.625,A -85,B 0,C 180,E1 -9332.928,E2 -9332.928} C_VEL
LIN {X 0,Y 432.375,Z 58.624,A -85,B 0,C 180,E1 -9336.023,E2 -9336.023} C_VEL
LIN {X 0,Y 432.353,Z 58.627,A -85,B 0,C 180,E1 -9339.046,E2 -9339.046} C_VEL
LIN {X 0,Y 432.38,Z 58.624,A -85,B 0,C 180,E1 -9342.011,E2 -9342.011} C_VEL
LIN {X 0,Y 432.398,Z 58.621,A -85,B 0,C 180,E1 -9344.926,E2 -9344.926} C_VEL
LIN {X 0,Y 432.462,Z 58.614,A -85,B 0,C 180,E1 -9347.803,E2 -9347.803} C_VEL
LIN {X 0,Y 432.494,Z 58.61,A -85,B 0,C 180,E1 -9351.59,E2 -9351.59} C_VEL
LIN {X 0,Y 432.597,Z 58.597,A -85,B 0,C 180,E1 -9354.406,E2 -9354.406} C_VEL
LIN {X 0,Y 432.605,Z 58.598,A -85,B 0,C 180,E1 -9358.138,E2 -9358.138} C_VEL
LIN {X 0,Y 432.734,Z 58.583,A -85,B 0,C 180,E1 -9360,E2 -9360} C_VEL
LIN {X 0,Y 432.593,Z 58.595,A -85,B 0,C 180,E1 -9362.793,E2 -9362.793} C_VEL
LIN {X 0,Y 432.593,Z 58.603,A -85,B 0,C 180,E1 -9365.594,E2 -9365.594} C_VEL
LIN {X 0,Y 432.466,Z 58.611,A -85,B 0,C 180,E1 -9368.41,E2 -9368.41} C_VEL
LIN {X 0,Y 432.461,Z 58.612,A -85,B 0,C 180,E1 -9372.196,E2 -9372.196} C_VEL
LIN {X 0,Y 432.432,Z 58.616,A -85,B 0,C 180,E1 -9376.039,E2 -9376.039} C_VEL
LIN {X 0,Y 432.388,Z 58.624,A -85,B 0,C 180,E1 -9379.485,E2 -9379.485} C_VEL
LIN {X 0,Y 432.32,Z 58.637,A -85,B 0,C 180,E1 -9382.964,E2 -9382.964} C_VEL
LIN {X 0,Y 432.345,Z 58.633,A -85,B 0,C 180,E1 -9385.002,E2 -9385.002} C_VEL
LIN {X 0,Y 432.382,Z 58.622,A -85,B 0,C 180,E1 -9388.123,E2 -9388.123} C_VEL
LIN {X 0,Y 432.323,Z 58.63,A -85,B 0,C 180,E1 -9391.346,E2 -9391.346} C_VEL
LIN {X 0,Y 432.342,Z 58.633,A -85,B 0,C 180,E1 -9394.677,E2 -9394.677} C_VEL
LIN {X 0,Y 432.337,Z 58.631,A -85,B 0,C 180,E1 -9398.15,E2 -9398.15} C_VEL
LIN {X 0,Y 432.334,Z 58.628,A -85,B 0,C 180,E1 -9401.602,E2 -9401.602} C_VEL
LIN {X 0,Y 432.335,Z 58.633,A -85,B 0,C 180,E1 -9404.347,E2 -9404.347} C_VEL
LIN {X 0,Y 432.321,Z 58.629,A -85,B 0,C 180,E1 -9407.016,E2 -9407.016} C_VEL
LIN {X 0,Y 432.335,Z 58.632,A -85,B 0,C 180,E1 -9409.821,E2 -9409.821} C_VEL
LIN {X 0,Y 432.308,Z 58.631,A -85,B 0,C 180,E1 -9413.022,E2 -9413.022} C_VEL
LIN {X 0,Y 432.361,Z 58.629,A -85,B 0,C 180,E1 -9415.996,E2 -9415.996} C_VEL
LIN {X 0,Y 432.349,Z 58.63,A -85,B 0,C 180,E1 -9419.489,E2 -9419.489} C_VEL
LIN {X 0,Y 432.468,Z 58.75,A -85,B 0,C 180,E1 -9422.409,E2 -9422.409} C_VEL
LIN {X 0,Y 434.892,Z 71.303,A -85,B 0,C 180,E1 -9424.821,E2 -9424.821} C_VEL
LIN {X 0,Y 434.704,Z 78.767,A -85,B 0,C 180,E1 -9426.16,E2 -9426.16} C_VEL
LIN {X 0,Y 434.009,Z 92.741,A -85,B 0,C 180,E1 -9428.632,E2 -9428.632} C_VEL
LIN {X 0,Y 433.115,Z 111.078,A -85,B 0,C 180,E1 -9431.844,E2 -9431.844} C_VEL
LIN {X 0,Y 436.627,Z 137.941,A -85,B 0,C 180,E1 -9432.428,E2 -9432.428} C_VEL
LIN {X 0,Y 435.798,Z 219.514,A -85,B 0,C 180,E1 -9433.788,E2 -9433.788} C_VEL
LIN {X 0,Y 435.36,Z 232.986,A -85,B 0,C 180,E1 -9434.192,E2 -9434.192} C_VEL
LIN {X 0,Y 434.811,Z 245.842,A -85,B 0,C 180,E1 -9434.772,E2 -9434.772} C_VEL
LIN {X 0,Y 434.181,Z 257.25,A -85,B 0,C 180,E1 -9435.469,E2 -9435.469} C_VEL
LIN {X 0,Y 433.579,Z 268.883,A -85,B 0,C 180,E1 -9436.394,E2 -9436.394} C_VEL
LIN {X 0,Y 432.954,Z 279.595,A -85,B 0,C 180,E1 -9437.46,E2 -9437.46} C_VEL
LIN {X 0,Y 432.472,Z 288.238,A -85,B 0,C 180,E1 -9438.517,E2 -9438.517} C_VEL
LIN {X 0,Y 431.969,Z 296.197,A -85,B 0,C 180,E1 -9439.69,E2 -9439.69} C_VEL
LIN {X 0,Y 431.608,Z 303.969,A -85,B 0,C 180,E1 -9441.101,E2 -9441.101} C_VEL
LIN {X 0,Y 431.414,Z 310.208,A -85,B 0,C 180,E1 -9442.511,E2 -9442.511} C_VEL
LIN {X 0,Y 431.25,Z 314.716,A -85,B 0,C 180,E1 -9443.778,E2 -9443.778} C_VEL
LIN {X 0,Y 431.277,Z 318.959,A -85,B 0,C 180,E1 -9445.326,E2 -9445.326} C_VEL
LIN {X 0,Y 431.255,Z 320.915,A -85,B 0,C 180,E1 -9446.262,E2 -9446.262} C_VEL
LIN {X 0,Y 431.329,Z 322.452,A -85,B 0,C 180,E1 -9447.198,E2 -9447.198} C_VEL
LIN {X 0,Y 431.29,Z 323.523,A -85,B 0,C 180,E1 -9448.132,E2 -9448.132} C_VEL
LIN {X 0,Y 431.289,Z 324.196,A -85,B 0,C 180,E1 -9449.066,E2 -9449.066} C_VEL
LIN {X 0,Y 431.297,Z 324.479,A -85,B 0,C 180,E1 -9450,E2 -9450} C_VEL
LIN {X 0,Y 431.259,Z 324.366,A -85,B 0,C 180,E1 -9450.933,E2 -9450.933} C_VEL
LIN {X 0,Y 431.269,Z 323.822,A -85,B 0,C 180,E1 -9451.867,E2 -9451.867} C_VEL
LIN {X 0,Y 431.325,Z 322.88,A -85,B 0,C 180,E1 -9452.801,E2 -9452.801} C_VEL
LIN {X 0,Y 431.27,Z 319.784,A -85,B 0,C 180,E1 -9454.673,E2 -9454.673} C_VEL
LIN {X 0,Y 431.249,Z 315.866,A -85,B 0,C 180,E1 -9456.222,E2 -9456.222} C_VEL
LIN {X 0,Y 431.436,Z 311.704,A -85,B 0,C 180,E1 -9457.488,E2 -9457.488} C_VEL
LIN {X 0,Y 431.72,Z 304.788,A -85,B 0,C 180,E1 -9459.132,E2 -9459.132} C_VEL
LIN {X 0,Y 432.157,Z 297.315,A -85,B 0,C 180,E1 -9460.542,E2 -9460.542} C_VEL
LIN {X 0,Y 432.779,Z 289.723,A -85,B 0,C 180,E1 -9461.712,E2 -9461.712} C_VEL
LIN {X 0,Y 433.34,Z 280.549,A -85,B 0,C 180,E1 -9462.885,E2 -9462.885} C_VEL
LIN {X 0,Y 434.045,Z 270.154,A -85,B 0,C 180,E1 -9463.959,E2 -9463.959} C_VEL
LIN {X 0,Y 434.836,Z 259.17,A -85,B 0,C 180,E1 -9464.867,E2 -9464.867} C_VEL
LIN {X 0,Y 435.638,Z 246.585,A -85,B 0,C 180,E1 -9465.677,E2 -9465.677} C_VEL
LIN {X 0,Y 436.306,Z 233.609,A -85,B 0,C 180,E1 -9466.282,E2 -9466.282} C_VEL
LIN {X 0,Y 436.929,Z 219.725,A -85,B 0,C 180,E1 -9466.709,E2 -9466.709} C_VEL
LIN {X 0,Y 437.824,Z 137.603,A -85,B 0,C 180,E1 -9468.106,E2 -9468.106} C_VEL
LIN {X 0,Y 434.97,Z 118.15,A -85,B 0,C 180,E1 -9468.584,E2 -9468.584} C_VEL
LIN {X 0,Y 433.642,Z 110.562,A -85,B 0,C 180,E1 -9468.792,E2 -9468.792} C_VEL
LIN {X 0,Y 434.706,Z 92.272,A -85,B 0,C 180,E1 -9472.079,E2 -9472.079} C_VEL
LIN {X 0,Y 435.766,Z 75.006,A -85,B 0,C 180,E1 -9475.244,E2 -9475.244} C_VEL
LIN {X 0,Y 433.637,Z 63.879,A -85,B 0,C 180,E1 -9477.509,E2 -9477.509} C_VEL
LIN {X 0,Y 432.376,Z 58.628,A -85,B 0,C 180,E1 -9478.629,E2 -9478.629} C_VEL
LIN {X 0,Y 432.321,Z 58.637,A -85,B 0,C 180,E1 -9481.346,E2 -9481.346} C_VEL
LIN {X 0,Y 432.34,Z 58.628,A -85,B 0,C 180,E1 -9484.677,E2 -9484.677} C_VEL
LIN {X 0,Y 432.346,Z 58.631,A -85,B 0,C 180,E1 -9488.148,E2 -9488.148} C_VEL
LIN {X 0,Y 432.332,Z 58.635,A -85,B 0,C 180,E1 -9491.602,E2 -9491.602} C_VEL
LIN {X 0,Y 432.332,Z 58.627,A -85,B 0,C 180,E1 -9494.347,E2 -9494.347} C_VEL
LIN {X 0,Y 432.318,Z 58.628,A -85,B 0,C 180,E1 -9497.015,E2 -9497.015} C_VEL
LIN {X 0,Y 432.355,Z 58.629,A -85,B 0,C 180,E1 -9499.817,E2 -9499.817} C_VEL
LIN {X 0,Y 432.315,Z 58.631,A -85,B 0,C 180,E1 -9503.023,E2 -9503.023} C_VEL
LIN {X 0,Y 432.357,Z 58.624,A -85,B 0,C 180,E1 -9505.996,E2 -9505.996} C_VEL
LIN {X 0,Y 432.345,Z 58.627,A -85,B 0,C 180,E1 -9509.489,E2 -9509.489} C_VEL
LIN {X 0,Y 432.39,Z 58.622,A -85,B 0,C 180,E1 -9512.928,E2 -9512.928} C_VEL
LIN {X 0,Y 432.369,Z 58.625,A -85,B 0,C 180,E1 -9516.023,E2 -9516.023} C_VEL
LIN {X 0,Y 432.348,Z 58.629,A -85,B 0,C 180,E1 -9519.046,E2 -9519.046} C_VEL
LIN {X 0,Y 432.376,Z 58.622,A -85,B 0,C 180,E1 -9522.011,E2 -9522.011} C_VEL
LIN {X 0,Y 432.393,Z 58.622,A -85,B 0,C 180,E1 -9524.927,E2 -9524.927} C_VEL
LIN {X 0,Y 432.457,Z 58.608,A -85,B 0,C 180,E1 -9527.804,E2 -9527.804} C_VEL
LIN {X 0,Y 432.49,Z 58.609,A -85,B 0,C 180,E1 -9531.59,E2 -9531.59} C_VEL
LIN {X 0,Y 432.592,Z 58.599,A -85,B 0,C 180,E1 -9534.406,E2 -9534.406} C_VEL
LIN {X 0,Y 432.6,Z 58.595,A -85,B 0,C 180,E1 -9538.138,E2 -9538.138} C_VEL
LIN {X 0,Y 432.729,Z 58.583,A -85,B 0,C 180,E1 -9540,E2 -9540} C_VEL
LIN {X 0,Y 432.589,Z 58.59,A -85,B 0,C 180,E1 -9542.794,E2 -9542.794} C_VEL
LIN {X 0,Y 432.589,Z 58.602,A -85,B 0,C 180,E1 -9545.594,E2 -9545.594} C_VEL
LIN {X 0,Y 432.461,Z 58.607,A -85,B 0,C 180,E1 -9548.411,E2 -9548.411} C_VEL
LIN {X 0,Y 432.457,Z 58.61,A -85,B 0,C 180,E1 -9552.197,E2 -9552.197} C_VEL
LIN {X 0,Y 432.428,Z 58.616,A -85,B 0,C 180,E1 -9556.039,E2 -9556.039} C_VEL
LIN {X 0,Y 432.385,Z 58.624,A -85,B 0,C 180,E1 -9559.485,E2 -9559.485} C_VEL
LIN {X 0,Y 432.316,Z 58.636,A -85,B 0,C 180,E1 -9562.965,E2 -9562.965} C_VEL
LIN {X 0,Y 432.338,Z 58.627,A -85,B 0,C 180,E1 -9565.002,E2 -9565.002} C_VEL
LIN {X 0,Y 432.346,Z 58.63,A -85,B 0,C 180,E1 -9568.126,E2 -9568.126} C_VEL
LIN {X 0,Y 432.319,Z 58.631,A -85,B 0,C 180,E1 -9571.347,E2 -9571.347} C_VEL
LIN {X 0,Y 432.336,Z 58.629,A -85,B 0,C 180,E1 -9574.678,E2 -9574.678} C_VEL
LIN {X 0,Y 432.328,Z 58.635,A -85,B 0,C 180,E1 -9578.151,E2 -9578.151} C_VEL
LIN {X 0,Y 432.311,Z 58.628,A -85,B 0,C 180,E1 -9581.599,E2 -9581.599} C_VEL
LIN {X 0,Y 432.333,Z 58.63,A -85,B 0,C 180,E1 -9584.348,E2 -9584.348} C_VEL
LIN {X 0,Y 432.307,Z 58.638,A -85,B 0,C 180,E1 -9587.018,E2 -9587.018} C_VEL
LIN {X 0,Y 432.289,Z 58.639,A -85,B 0,C 180,E1 -9589.829,E2 -9589.829} C_VEL
LIN {X 0,Y 432.3,Z 58.638,A -85,B 0,C 180,E1 -9593.022,E2 -9593.022} C_VEL
LIN {X 0,Y 432.385,Z 58.741,A -85,B 0,C 180,E1 -9594.902,E2 -9594.902} C_VEL
LIN {X 0,Y 434.196,Z 68.153,A -85,B 0,C 180,E1 -9597.294,E2 -9597.294} C_VEL
LIN {X 0,Y 437.76,Z 81.547,A -85,B 0,C 180,E1 -9597.714,E2 -9597.714} C_VEL
LIN {X 0,Y 438.48,Z 85.663,A -85,B 0,C 180,E1 -9597.822,E2 -9597.822} C_VEL
LIN {X 0,Y 437.352,Z 174.469,A -85,B 0,C 180,E1 -9599.323,E2 -9599.323} C_VEL
LIN {X 0,Y 436.975,Z 187.623,A -85,B 0,C 180,E1 -9599.728,E2 -9599.728} C_VEL
LIN {X 0,Y 436.573,Z 200.133,A -85,B 0,C 180,E1 -9600.307,E2 -9600.307} C_VEL
LIN {X 0,Y 435.956,Z 212.396,A -85,B 0,C 180,E1 -9601.078,E2 -9601.078} C_VEL
LIN {X 0,Y 435.232,Z 223.125,A -85,B 0,C 180,E1 -9601.947,E2 -9601.947} C_VEL
LIN {X 0,Y 434.499,Z 234.152,A -85,B 0,C 180,E1 -9603.071,E2 -9603.071} C_VEL
LIN {X 0,Y 433.784,Z 243.893,A -85,B 0,C 180,E1 -9604.317,E2 -9604.317} C_VEL
LIN {X 0,Y 433.172,Z 252.208,A -85,B 0,C 180,E1 -9605.636,E2 -9605.636} C_VEL
LIN {X 0,Y 432.589,Z 259.444,A -85,B 0,C 180,E1 -9607.051,E2 -9607.051} C_VEL
LIN {X 0,Y 432.158,Z 265.478,A -85,B 0,C 180,E1 -9608.537,E2 -9608.537} C_VEL
LIN {X 0,Y 431.858,Z 270.126,A -85,B 0,C 180,E1 -9610.017,E2 -9610.017} C_VEL
LIN {X 0,Y 431.655,Z 272.544,A -85,B 0,C 180,E1 -9610.997,E2 -9610.997} C_VEL
LIN {X 0,Y 431.452,Z 274.502,A -85,B 0,C 180,E1 -9611.972,E2 -9611.972} C_VEL
LIN {X 0,Y 431.373,Z 275.976,A -85,B 0,C 180,E1 -9612.947,E2 -9612.947} C_VEL
LIN {X 0,Y 431.258,Z 277.498,A -85,B 0,C 180,E1 -9614.708,E2 -9614.708} C_VEL
LIN {X 0,Y 430.591,Z 277.847,A -85,B 0,C 180,E1 -9615.487,E2 -9615.487} C_VEL
LIN {X 0,Y 427.742,Z 277.84,A -85,B 0,C 180,E1 -9616.755,E2 -9616.755} C_VEL
LIN {X 0,Y 425.345,Z 277.247,A -85,B 0,C 180,E1 -9617.775,E2 -9617.775} C_VEL
LIN {X 0,Y 424.33,Z 276.441,A -85,B 0,C 180,E1 -9618.557,E2 -9618.557} C_VEL
LIN {X 0,Y 424.255,Z 276.066,A -85,B 0,C 180,E1 -9618.82,E2 -9618.82} C_VEL
LIN {X 0,Y 424.397,Z 273.26,A -85,B 0,C 180,E1 -9620.468,E2 -9620.468} C_VEL
LIN {X 0,Y 424.594,Z 269.669,A -85,B 0,C 180,E1 -9621.912,E2 -9621.912} C_VEL
LIN {X 0,Y 424.841,Z 264.968,A -85,B 0,C 180,E1 -9623.351,E2 -9623.351} C_VEL
LIN {X 0,Y 425.147,Z 259.027,A -85,B 0,C 180,E1 -9624.784,E2 -9624.784} C_VEL
LIN {X 0,Y 425.598,Z 251.631,A -85,B 0,C 180,E1 -9626.213,E2 -9626.213} C_VEL
LIN {X 0,Y 426.134,Z 244.081,A -85,B 0,C 180,E1 -9627.401,E2 -9627.401} C_VEL
LIN {X 0,Y 426.753,Z 234.951,A -85,B 0,C 180,E1 -9628.585,E2 -9628.585} C_VEL
LIN {X 0,Y 427.341,Z 224.816,A -85,B 0,C 180,E1 -9629.647,E2 -9629.647} C_VEL
LIN {X 0,Y 427.978,Z 213.569,A -85,B 0,C 180,E1 -9630.588,E2 -9630.588} C_VEL
LIN {X 0,Y 428.487,Z 201.947,A -85,B 0,C 180,E1 -9631.351,E2 -9631.351} C_VEL
LIN {X 0,Y 428.819,Z 189.325,A -85,B 0,C 180,E1 -9631.968,E2 -9631.968} C_VEL
LIN {X 0,Y 429.179,Z 175.835,A -85,B 0,C 180,E1 -9632.406,E2 -9632.406} C_VEL
LIN {X 0,Y 429.651,Z 134.137,A -85,B 0,C 180,E1 -9633.136,E2 -9633.136} C_VEL
LIN {X 0,Y 430.042,Z 84.584,A -85,B 0,C 180,E1 -9633.97,E2 -9633.97} C_VEL
LIN {X 0,Y 426.689,Z 67.887,A -85,B 0,C 180,E1 -9634.399,E2 -9634.399} C_VEL
LIN {X 0,Y 425.549,Z 59.481,A -85,B 0,C 180,E1 -9636.46,E2 -9636.46} C_VEL
LIN {X 0,Y 425.448,Z 59.493,A -85,B 0,C 180,E1 -9638.55,E2 -9638.55} C_VEL
LIN {X 0,Y 425.418,Z 59.495,A -85,B 0,C 180,E1 -9642.402,E2 -9642.402} C_VEL
LIN {X 0,Y 425.393,Z 59.499,A -85,B 0,C 180,E1 -9646.312,E2 -9646.312} C_VEL
LIN {X 0,Y 425.334,Z 59.501,A -85,B 0,C 180,E1 -9649.636,E2 -9649.636} C_VEL
LIN {X 0,Y 425.293,Z 59.51,A -85,B 0,C 180,E1 -9652.339,E2 -9652.339} C_VEL
LIN {X 0,Y 425.296,Z 59.505,A -85,B 0,C 180,E1 -9655.446,E2 -9655.446} C_VEL
LIN {X 0,Y 425.354,Z 59.5,A -85,B 0,C 180,E1 -9657.558,E2 -9657.558} C_VEL
LIN {X 0,Y 425.293,Z 59.505,A -85,B 0,C 180,E1 -9660.816,E2 -9660.816} C_VEL
LIN {X 0,Y 425.317,Z 59.503,A -85,B 0,C 180,E1 -9664.288,E2 -9664.288} C_VEL
LIN {X 0,Y 425.29,Z 59.512,A -85,B 0,C 180,E1 -9667.693,E2 -9667.693} C_VEL
LIN {X 0,Y 425.288,Z 59.505,A -85,B 0,C 180,E1 -9670.521,E2 -9670.521} C_VEL
LIN {X 0,Y 425.262,Z 59.515,A -85,B 0,C 180,E1 -9673.351,E2 -9673.351} C_VEL
LIN {X 0,Y 425.261,Z 59.51,A -85,B 0,C 180,E1 -9676.649,E2 -9676.649} C_VEL
LIN {X 0,Y 425.29,Z 59.506,A -85,B 0,C 180,E1 -9679.873,E2 -9679.873} C_VEL
LIN {X 0,Y 425.282,Z 59.507,A -85,B 0,C 180,E1 -9682.488,E2 -9682.488} C_VEL
LIN {X 0,Y 425.311,Z 59.503,A -85,B 0,C 180,E1 -9685.817,E2 -9685.817} C_VEL
LIN {X 0,Y 425.294,Z 59.508,A -85,B 0,C 180,E1 -9689.239,E2 -9689.239} C_VEL
LIN {X 0,Y 425.352,Z 59.501,A -85,B 0,C 180,E1 -9692.442,E2 -9692.442} C_VEL
LIN {X 0,Y 425.355,Z 59.497,A -85,B 0,C 180,E1 -9695.602,E2 -9695.602} C_VEL
LIN {X 0,Y 425.297,Z 59.51,A -85,B 0,C 180,E1 -9698.681,E2 -9698.681} C_VEL
LIN {X 0,Y 425.336,Z 59.5,A -85,B 0,C 180,E1 -9701.703,E2 -9701.703} C_VEL
LIN {X 0,Y 425.351,Z 59.501,A -85,B 0,C 180,E1 -9704.67,E2 -9704.67} C_VEL
LIN {X 0,Y 425.415,Z 59.491,A -85,B 0,C 180,E1 -9707.598,E2 -9707.598} C_VEL
LIN {X 0,Y 425.445,Z 59.487,A -85,B 0,C 180,E1 -9711.45,E2 -9711.45} C_VEL
LIN {X 0,Y 425.553,Z 59.476,A -85,B 0,C 180,E1 -9714.313,E2 -9714.313} C_VEL
LIN {X 0,Y 425.575,Z 59.474,A -85,B 0,C 180,E1 -9718.107,E2 -9718.107} C_VEL
LIN {X 0,Y 425.703,Z 59.458,A -85,B 0,C 180,E1 -9720,E2 -9720} C_VEL
LIN {X 0,Y 425.547,Z 59.473,A -85,B 0,C 180,E1 -9722.84,E2 -9722.84} C_VEL
LIN {X 0,Y 425.549,Z 59.479,A -85,B 0,C 180,E1 -9725.687,E2 -9725.687} C_VEL
LIN {X 0,Y 425.41,Z 59.49,A -85,B 0,C 180,E1 -9728.551,E2 -9728.551} C_VEL
LIN {X 0,Y 425.414,Z 59.49,A -85,B 0,C 180,E1 -9732.402,E2 -9732.402} C_VEL
LIN {X 0,Y 425.39,Z 59.493,A -85,B 0,C 180,E1 -9736.312,E2 -9736.312} C_VEL
LIN {X 0,Y 425.33,Z 59.502,A -85,B 0,C 180,E1 -9739.635,E2 -9739.635} C_VEL
LIN {X 0,Y 425.29,Z 59.506,A -85,B 0,C 180,E1 -9742.339,E2 -9742.339} C_VEL
LIN {X 0,Y 425.324,Z 59.505,A -85,B 0,C 180,E1 -9744.658,E2 -9744.658} C_VEL
LIN {X 0,Y 425.347,Z 59.498,A -85,B 0,C 180,E1 -9747.558,E2 -9747.558} C_VEL
LIN {X 0,Y 425.289,Z 59.511,A -85,B 0,C 180,E1 -9750.816,E2 -9750.816} C_VEL
LIN {X 0,Y 425.313,Z 59.506,A -85,B 0,C 180,E1 -9754.288,E2 -9754.288} C_VEL
LIN {X 0,Y 425.28,Z 59.507,A -85,B 0,C 180,E1 -9757.694,E2 -9757.694} C_VEL
LIN {X 0,Y 425.281,Z 59.512,A -85,B 0,C 180,E1 -9760.52,E2 -9760.52} C_VEL
LIN {X 0,Y 425.258,Z 59.509,A -85,B 0,C 180,E1 -9763.351,E2 -9763.351} C_VEL
LIN {X 0,Y 425.259,Z 59.511,A -85,B 0,C 180,E1 -9766.649,E2 -9766.649} C_VEL
LIN {X 0,Y 425.289,Z 59.51,A -85,B 0,C 180,E1 -9769.873,E2 -9769.873} C_VEL
LIN {X 0,Y 425.28,Z 59.508,A -85,B 0,C 180,E1 -9772.488,E2 -9772.488} C_VEL
LIN {X 0,Y 425.31,Z 59.51,A -85,B 0,C 180,E1 -9775.817,E2 -9775.817} C_VEL
LIN {X 0,Y 425.293,Z 59.507,A -85,B 0,C 180,E1 -9779.239,E2 -9779.239} C_VEL
LIN {X 0,Y 425.441,Z 59.66,A -85,B 0,C 180,E1 -9782.215,E2 -9782.215} C_VEL
LIN {X 0,Y 427.912,Z 72.471,A -85,B 0,C 180,E1 -9784.721,E2 -9784.721} C_VEL
LIN {X 0,Y 427.75,Z 79.515,A -85,B 0,C 180,E1 -9786.005,E2 -9786.005} C_VEL
LIN {X 0,Y 426.999,Z 93.492,A -85,B 0,C 180,E1 -9788.517,E2 -9788.517} C_VEL
LIN {X 0,Y 426.123,Z 110.739,A -85,B 0,C 180,E1 -9791.59,E2 -9791.59} C_VEL
LIN {X 0,Y 429.774,Z 138.594,A -85,B 0,C 180,E1 -9792.201,E2 -9792.201} C_VEL
LIN {X 0,Y 428.879,Z 219.844,A -85,B 0,C 180,E1 -9793.58,E2 -9793.58} C_VEL
LIN {X 0,Y 428.442,Z 233.077,A -85,B 0,C 180,E1 -9793.991,E2 -9793.991} C_VEL
LIN {X 0,Y 427.885,Z 245.823,A -85,B 0,C 180,E1 -9794.58,E2 -9794.58} C_VEL
LIN {X 0,Y 427.164,Z 257.931,A -85,B 0,C 180,E1 -9795.347,E2 -9795.347} C_VEL
LIN {X 0,Y 426.535,Z 269.518,A -85,B 0,C 180,E1 -9796.299,E2 -9796.299} C_VEL
LIN {X 0,Y 425.913,Z 279.938,A -85,B 0,C 180,E1 -9797.371,E2 -9797.371} C_VEL
LIN {X 0,Y 425.357,Z 289.288,A -85,B 0,C 180,E1 -9798.564,E2 -9798.564} C_VEL
LIN {X 0,Y 424.789,Z 298.358,A -85,B 0,C 180,E1 -9799.996,E2 -9799.996} C_VEL
LIN {X 0,Y 424.5,Z 305.668,A -85,B 0,C 180,E1 -9801.431,E2 -9801.431} C_VEL
LIN {X 0,Y 424.313,Z 311.498,A -85,B 0,C 180,E1 -9802.864,E2 -9802.864} C_VEL
LIN {X 0,Y 424.157,Z 316.074,A -85,B 0,C 180,E1 -9804.294,E2 -9804.294} C_VEL
LIN {X 0,Y 424.206,Z 318.489,A -85,B 0,C 180,E1 -9805.248,E2 -9805.248} C_VEL
LIN {X 0,Y 424.161,Z 320.458,A -85,B 0,C 180,E1 -9806.2,E2 -9806.2} C_VEL
LIN {X 0,Y 424.257,Z 322.015,A -85,B 0,C 180,E1 -9807.151,E2 -9807.151} C_VEL
LIN {X 0,Y 424.212,Z 323.107,A -85,B 0,C 180,E1 -9808.101,E2 -9808.101} C_VEL
LIN {X 0,Y 424.202,Z 323.792,A -85,B 0,C 180,E1 -9809.05,E2 -9809.05} C_VEL
LIN {X 0,Y 424.207,Z 324.087,A -85,B 0,C 180,E1 -9810,E2 -9810} C_VEL
LIN {X 0,Y 424.174,Z 323.99,A -85,B 0,C 180,E1 -9810.949,E2 -9810.949} C_VEL
LIN {X 0,Y 424.193,Z 323.469,A -85,B 0,C 180,E1 -9811.899,E2 -9811.899} C_VEL
LIN {X 0,Y 424.234,Z 322.538,A -85,B 0,C 180,E1 -9812.848,E2 -9812.848} C_VEL
LIN {X 0,Y 424.195,Z 319.471,A -85,B 0,C 180,E1 -9814.751,E2 -9814.751} C_VEL
LIN {X 0,Y 424.151,Z 315.981,A -85,B 0,C 180,E1 -9816.186,E2 -9816.186} C_VEL
LIN {X 0,Y 424.361,Z 311.443,A -85,B 0,C 180,E1 -9817.613,E2 -9817.613} C_VEL
LIN {X 0,Y 424.678,Z 304.576,A -85,B 0,C 180,E1 -9819.285,E2 -9819.285} C_VEL
LIN {X 0,Y 425.158,Z 297.151,A -85,B 0,C 180,E1 -9820.717,E2 -9820.717} C_VEL
LIN {X 0,Y 425.904,Z 287.958,A -85,B 0,C 180,E1 -9822.145,E2 -9822.145} C_VEL
LIN {X 0,Y 426.602,Z 277.594,A -85,B 0,C 180,E1 -9823.429,E2 -9823.429} C_VEL
LIN {X 0,Y 427.459,Z 266.609,A -85,B 0,C 180,E1 -9824.52,E2 -9824.52} C_VEL
LIN {X 0,Y 428.17,Z 256.192,A -85,B 0,C 180,E1 -9825.347,E2 -9825.347} C_VEL
LIN {X 0,Y 429.03,Z 243.696,A -85,B 0,C 180,E1 -9826.108,E2 -9826.108} C_VEL
LIN {X 0,Y 429.748,Z 230.552,A -85,B 0,C 180,E1 -9826.691,E2 -9826.691} C_VEL
LIN {X 0,Y 430.26,Z 217.322,A -85,B 0,C 180,E1 -9827.068,E2 -9827.068} C_VEL
LIN {X 0,Y 431.074,Z 137.59,A -85,B 0,C 180,E1 -9828.44,E2 -9828.44} C_VEL
LIN {X 0,Y 428.266,Z 118.581,A -85,B 0,C 180,E1 -9828.92,E2 -9828.92} C_VEL
LIN {X 0,Y 426.756,Z 110.095,A -85,B 0,C 180,E1 -9829.167,E2 -9829.167} C_VEL
LIN {X 0,Y 427.865,Z 92.221,A -85,B 0,C 180,E1 -9832.442,E2 -9832.442} C_VEL
LIN {X 0,Y 428.875,Z 77.321,A -85,B 0,C 180,E1 -9835.218,E2 -9835.218} C_VEL
LIN {X 0,Y 428.134,Z 71.924,A -85,B 0,C 180,E1 -9836.309,E2 -9836.309} C_VEL
LIN {X 0,Y 425.677,Z 61.127,A -85,B 0,C 180,E1 -9838.606,E2 -9838.606} C_VEL
LIN {X 0,Y 425.304,Z 59.509,A -85,B 0,C 180,E1 -9839.009,E2 -9839.009} C_VEL
LIN {X 0,Y 425.265,Z 59.518,A -85,B 0,C 180,E1 -9841.926,E2 -9841.926} C_VEL
LIN {X 0,Y 425.3,Z 59.504,A -85,B 0,C 180,E1 -9845.335,E2 -9845.335} C_VEL
LIN {X 0,Y 425.302,Z 59.506,A -85,B 0,C 180,E1 -9849.044,E2 -9849.044} C_VEL
LIN {X 0,Y 425.273,Z 59.509,A -85,B 0,C 180,E1 -9852.653,E2 -9852.653} C_VEL
LIN {X 0,Y 425.259,Z 59.505,A -85,B 0,C 180,E1 -9856.044,E2 -9856.044} C_VEL
LIN {X 0,Y 425.303,Z 59.505,A -85,B 0,C 180,E1 -9858.625,E2 -9858.625} C_VEL
LIN {X 0,Y 425.322,Z 59.506,A -85,B 0,C 180,E1 -9861.104,E2 -9861.104} C_VEL
LIN {X 0,Y 425.299,Z 59.507,A -85,B 0,C 180,E1 -9864.664,E2 -9864.664} C_VEL
LIN {X 0,Y 425.263,Z 59.51,A -85,B 0,C 180,E1 -9868.073,E2 -9868.073} C_VEL
LIN {X 0,Y 425.329,Z 59.503,A -85,B 0,C 180,E1 -9871.368,E2 -9871.368} C_VEL
LIN {X 0,Y 425.293,Z 59.506,A -85,B 0,C 180,E1 -9874.555,E2 -9874.555} C_VEL
LIN {X 0,Y 425.285,Z 59.5,A -85,B 0,C 180,E1 -9877.661,E2 -9877.661} C_VEL
LIN {X 0,Y 425.362,Z 59.498,A -85,B 0,C 180,E1 -9880.704,E2 -9880.704} C_VEL
LIN {X 0,Y 425.386,Z 59.493,A -85,B 0,C 180,E1 -9883.688,E2 -9883.688} C_VEL
LIN {X 0,Y 425.409,Z 59.484,A -85,B 0,C 180,E1 -9887.598,E2 -9887.598} C_VEL
LIN {X 0,Y 425.44,Z 59.486,A -85,B 0,C 180,E1 -9891.45,E2 -9891.45} C_VEL
LIN {X 0,Y 425.549,Z 59.477,A -85,B 0,C 180,E1 -9894.313,E2 -9894.313} C_VEL
LIN {X 0,Y 425.57,Z 59.47,A -85,B 0,C 180,E1 -9898.107,E2 -9898.107} C_VEL
LIN {X 0,Y 425.699,Z 59.459,A -85,B 0,C 180,E1 -9900,E2 -9900} C_VEL
LIN {X 0,Y 425.542,Z 59.468,A -85,B 0,C 180,E1 -9902.84,E2 -9902.84} C_VEL
LIN {X 0,Y 425.544,Z 59.478,A -85,B 0,C 180,E1 -9905.687,E2 -9905.687} C_VEL
LIN {X 0,Y 425.406,Z 59.486,A -85,B 0,C 180,E1 -9908.551,E2 -9908.551} C_VEL
LIN {X 0,Y 425.41,Z 59.488,A -85,B 0,C 180,E1 -9912.402,E2 -9912.402} C_VEL
LIN {X 0,Y 425.386,Z 59.494,A -85,B 0,C 180,E1 -9916.312,E2 -9916.312} C_VEL
LIN {X 0,Y 425.326,Z 59.503,A -85,B 0,C 180,E1 -9919.636,E2 -9919.636} C_VEL
LIN {X 0,Y 425.286,Z 59.503,A -85,B 0,C 180,E1 -9922.339,E2 -9922.339} C_VEL
LIN {X 0,Y 425.319,Z 59.506,A -85,B 0,C 180,E1 -9924.658,E2 -9924.658} C_VEL
LIN {X 0,Y 425.298,Z 59.506,A -85,B 0,C 180,E1 -9927.562,E2 -9927.562} C_VEL
LIN {X 0,Y 425.286,Z 59.51,A -85,B 0,C 180,E1 -9930.817,E2 -9930.817} C_VEL
LIN {X 0,Y 425.308,Z 59.509,A -85,B 0,C 180,E1 -9934.288,E2 -9934.288} C_VEL
LIN {X 0,Y 425.275,Z 59.511,A -85,B 0,C 180,E1 -9937.695,E2 -9937.695} C_VEL
LIN {X 0,Y 425.254,Z 59.507,A -85,B 0,C 180,E1 -9940.517,E2 -9940.517} C_VEL
LIN {X 0,Y 425.258,Z 59.516,A -85,B 0,C 180,E1 -9943.957,E2 -9943.957} C_VEL
LIN {X 0,Y 425.249,Z 59.517,A -85,B 0,C 180,E1 -9946.651,E2 -9946.651} C_VEL
LIN {X 0,Y 425.243,Z 59.517,A -85,B 0,C 180,E1 -9949.868,E2 -9949.868} C_VEL
LIN {X 0,Y 425.272,Z 59.513,A -85,B 0,C 180,E1 -9952.49,E2 -9952.49} C_VEL
LIN {X 0,Y 425.305,Z 59.565,A -85,B 0,C 180,E1 -9954.592,E2 -9954.592} C_VEL
LIN {X 0,Y 427.167,Z 68.693,A -85,B 0,C 180,E1 -9956.922,E2 -9956.922} C_VEL
LIN {X 0,Y 430.106,Z 78.286,A -85,B 0,C 180,E1 -9957.254,E2 -9957.254} C_VEL
LIN {X 0,Y 431.891,Z 86.93,A -85,B 0,C 180,E1 -9957.504,E2 -9957.504} C_VEL
LIN {X 0,Y 430.643,Z 175.638,A -85,B 0,C 180,E1 -9959.031,E2 -9959.031} C_VEL
LIN {X 0,Y 430.278,Z 188.966,A -85,B 0,C 180,E1 -9959.461,E2 -9959.461} C_VEL
LIN {X 0,Y 429.827,Z 201.547,A -85,B 0,C 180,E1 -9960.066,E2 -9960.066} C_VEL
LIN {X 0,Y 429.167,Z 213.478,A -85,B 0,C 180,E1 -9960.845,E2 -9960.845} C_VEL
LIN {X 0,Y 428.408,Z 224.078,A -85,B 0,C 180,E1 -9961.726,E2 -9961.726} C_VEL
LIN {X 0,Y 427.64,Z 235.003,A -85,B 0,C 180,E1 -9962.868,E2 -9962.868} C_VEL
LIN {X 0,Y 426.869,Z 244.633,A -85,B 0,C 180,E1 -9964.133,E2 -9964.133} C_VEL
LIN {X 0,Y 426.29,Z 252.126,A -85,B 0,C 180,E1 -9965.337,E2 -9965.337} C_VEL
LIN {X 0,Y 425.601,Z 260.068,A -85,B 0,C 180,E1 -9966.91,E2 -9966.91} C_VEL
LIN {X 0,Y 425.177,Z 265.242,A -85,B 0,C 180,E1 -9968.199,E2 -9968.199} C_VEL
LIN {X 0,Y 424.86,Z 269.962,A -85,B 0,C 180,E1 -9969.673,E2 -9969.673} C_VEL
LIN {X 0,Y 424.544,Z 273.582,A -85,B 0,C 180,E1 -9971.168,E2 -9971.168} C_VEL
LIN {X 0,Y 424.324,Z 276.107,A -85,B 0,C 180,E1 -9972.655,E2 -9972.655} C_VEL
LIN {X 0,Y 424.23,Z 277.441,A -85,B 0,C 180,E1 -9973.918,E2 -9973.918} C_VEL
LIN {X 0,Y 424.14,Z 278.173,A -85,B 0,C 180,E1 -9975.609,E2 -9975.609} C_VEL
LIN {X 0,Y 424.155,Z 278.038,A -85,B 0,C 180,E1 -9976.587,E2 -9976.587} C_VEL
LIN {X 0,Y 424.236,Z 277.249,A -85,B 0,C 180,E1 -9977.801,E2 -9977.801} C_VEL
LIN {X 0,Y 424.255,Z 276.066,A -85,B 0,C 180,E1 -9978.82,E2 -9978.82} C_VEL
LIN {X 0,Y 423.633,Z 274.979,A -85,B 0,C 180,E1 -9979.599,E2 -9979.599} C_VEL
LIN {X 0,Y 420.911,Z 272.627,A -85,B 0,C 180,E1 -9980.855,E2 -9980.855} C_VEL
LIN {X 0,Y 418.647,Z 270.306,A -85,B 0,C 180,E1 -9981.849,E2 -9981.849} C_VEL
LIN {X 0,Y 417.736,Z 268.172,A -85,B 0,C 180,E1 -9982.597,E2 -9982.597} C_VEL
LIN {X 0,Y 417.695,Z 267.355,A -85,B 0,C 180,E1 -9982.846,E2 -9982.846} C_VEL
LIN {X 0,Y 417.935,Z 261.335,A -85,B 0,C 180,E1 -9984.452,E2 -9984.452} C_VEL
LIN {X 0,Y 418.417,Z 254.416,A -85,B 0,C 180,E1 -9985.907,E2 -9985.907} C_VEL
LIN {X 0,Y 419.054,Z 245.739,A -85,B 0,C 180,E1 -9987.357,E2 -9987.357} C_VEL
LIN {X 0,Y 419.655,Z 236.869,A -85,B 0,C 180,E1 -9988.561,E2 -9988.561} C_VEL
LIN {X 0,Y 420.252,Z 227.14,A -85,B 0,C 180,E1 -9989.641,E2 -9989.641} C_VEL
LIN {X 0,Y 420.935,Z 216.416,A -85,B 0,C 180,E1 -9990.598,E2 -9990.598} C_VEL
LIN {X 0,Y 421.494,Z 204.442,A -85,B 0,C 180,E1 -9991.434,E2 -9991.434} C_VEL
LIN {X 0,Y 421.873,Z 192.749,A -85,B 0,C 180,E1 -9992.054,E2 -9992.054} C_VEL
LIN {X 0,Y 422.225,Z 180.531,A -85,B 0,C 180,E1 -9992.515,E2 -9992.515} C_VEL
LIN {X 0,Y 422.439,Z 166.505,A -85,B 0,C 180,E1 -9992.831,E2 -9992.831} C_VEL
LIN {X 0,Y 423.307,Z 86.209,A -85,B 0,C 180,E1 -9994.197,E2 -9994.197} C_VEL
LIN {X 0,Y 419.671,Z 68.233,A -85,B 0,C 180,E1 -9994.668,E2 -9994.668} C_VEL
LIN {X 0,Y 418.512,Z 60.356,A -85,B 0,C 180,E1 -9996.63,E2 -9996.63} C_VEL
LIN {X 0,Y 418.406,Z 60.369,A -85,B 0,C 180,E1 -9998.695,E2 -9998.695} C_VEL
LIN {X 0,Y 418.361,Z 60.374,A -85,B 0,C 180,E1 -10002.615,E2 -10002.615} C_VEL
LIN {X 0,Y 418.307,Z 60.375,A -85,B 0,C 180,E1 -10005.594,E2 -10005.594} C_VEL
LIN {X 0,Y 418.287,Z 60.381,A -85,B 0,C 180,E1 -10008.617,E2 -10008.617} C_VEL
LIN {X 0,Y 418.239,Z 60.385,A -85,B 0,C 180,E1 -10011.696,E2 -10011.696} C_VEL
LIN {X 0,Y 418.289,Z 60.378,A -85,B 0,C 180,E1 -10014.864,E2 -10014.864} C_VEL
LIN {X 0,Y 418.296,Z 60.382,A -85,B 0,C 180,E1 -10018.063,E2 -10018.063} C_VEL
LIN {X 0,Y 418.217,Z 60.388,A -85,B 0,C 180,E1 -10021.396,E2 -10021.396} C_VEL
LIN {X 0,Y 418.271,Z 60.38,A -85,B 0,C 180,E1 -10024.58,E2 -10024.58} C_VEL
LIN {X 0,Y 418.239,Z 60.388,A -85,B 0,C 180,E1 -10027.834,E2 -10027.834} C_VEL
LIN {X 0,Y 418.228,Z 60.386,A -85,B 0,C 180,E1 -10030.948,E2 -10030.948} C_VEL
LIN {X 0,Y 418.214,Z 60.39,A -85,B 0,C 180,E1 -10033.729,E2 -10033.729} C_VEL
LIN {X 0,Y 418.212,Z 60.387,A -85,B 0,C 180,E1 -10036.448,E2 -10036.448} C_VEL
LIN {X 0,Y 418.227,Z 60.391,A -85,B 0,C 180,E1 -10039.13,E2 -10039.13} C_VEL
LIN {X 0,Y 418.232,Z 60.384,A -85,B 0,C 180,E1 -10042.166,E2 -10042.166} C_VEL
LIN {X 0,Y 418.269,Z 60.382,A -85,B 0,C 180,E1 -10045.42,E2 -10045.42} C_VEL
LIN {X 0,Y 418.215,Z 60.39,A -85,B 0,C 180,E1 -10048.604,E2 -10048.604} C_VEL
LIN {X 0,Y 418.295,Z 60.377,A -85,B 0,C 180,E1 -10051.936,E2 -10051.936} C_VEL
LIN {X 0,Y 418.293,Z 60.379,A -85,B 0,C 180,E1 -10055.162,E2 -10055.162} C_VEL
LIN {X 0,Y 418.238,Z 60.388,A -85,B 0,C 180,E1 -10058.303,E2 -10058.303} C_VEL
LIN {X 0,Y 418.286,Z 60.378,A -85,B 0,C 180,E1 -10061.383,E2 -10061.383} C_VEL
LIN {X 0,Y 418.306,Z 60.382,A -85,B 0,C 180,E1 -10064.406,E2 -10064.406} C_VEL
LIN {X 0,Y 418.358,Z 60.369,A -85,B 0,C 180,E1 -10067.385,E2 -10067.385} C_VEL
LIN {X 0,Y 418.403,Z 60.363,A -85,B 0,C 180,E1 -10071.305,E2 -10071.305} C_VEL
LIN {X 0,Y 418.512,Z 60.354,A -85,B 0,C 180,E1 -10074.217,E2 -10074.217} C_VEL
LIN {X 0,Y 418.544,Z 60.35,A -85,B 0,C 180,E1 -10078.075,E2 -10078.075} C_VEL
LIN {X 0,Y 418.673,Z 60.334,A -85,B 0,C 180,E1 -10080,E2 -10080} C_VEL
LIN {X 0,Y 418.502,Z 60.351,A -85,B 0,C 180,E1 -10082.888,E2 -10082.888} C_VEL
LIN {X 0,Y 418.507,Z 60.355,A -85,B 0,C 180,E1 -10085.783,E2 -10085.783} C_VEL
LIN {X 0,Y 418.38,Z 60.366,A -85,B 0,C 180,E1 -10088.695,E2 -10088.695} C_VEL
LIN {X 0,Y 418.318,Z 60.378,A -85,B 0,C 180,E1 -10091.631,E2 -10091.631} C_VEL
LIN {X 0,Y 418.305,Z 60.376,A -85,B 0,C 180,E1 -10094.597,E2 -10094.597} C_VEL
LIN {X 0,Y 418.288,Z 60.38,A -85,B 0,C 180,E1 -10097.604,E2 -10097.604} C_VEL
LIN {X 0,Y 418.252,Z 60.385,A -85,B 0,C 180,E1 -10100.663,E2 -10100.663} C_VEL
LIN {X 0,Y 418.277,Z 60.379,A -85,B 0,C 180,E1 -10103.782,E2 -10103.782} C_VEL
LIN {X 0,Y 418.312,Z 60.379,A -85,B 0,C 180,E1 -10107.07,E2 -10107.07} C_VEL
LIN {X 0,Y 418.246,Z 60.385,A -85,B 0,C 180,E1 -10110.272,E2 -10110.272} C_VEL
LIN {X 0,Y 418.25,Z 60.382,A -85,B 0,C 180,E1 -10113.677,E2 -10113.677} C_VEL
LIN {X 0,Y 418.241,Z 60.384,A -85,B 0,C 180,E1 -10117.224,E2 -10117.224} C_VEL
LIN {X 0,Y 418.246,Z 60.383,A -85,B 0,C 180,E1 -10119.683,E2 -10119.683} C_VEL
LIN {X 0,Y 418.231,Z 60.392,A -85,B 0,C 180,E1 -10122.321,E2 -10122.321} C_VEL
LIN {X 0,Y 418.237,Z 60.384,A -85,B 0,C 180,E1 -10125.109,E2 -10125.109} C_VEL
LIN {X 0,Y 418.242,Z 60.386,A -85,B 0,C 180,E1 -10127.767,E2 -10127.767} C_VEL
LIN {X 0,Y 418.254,Z 60.383,A -85,B 0,C 180,E1 -10130.619,E2 -10130.619} C_VEL
LIN {X 0,Y 418.245,Z 60.389,A -85,B 0,C 180,E1 -10133.976,E2 -10133.976} C_VEL
LIN {X 0,Y 418.26,Z 60.382,A -85,B 0,C 180,E1 -10137.156,E2 -10137.156} C_VEL
LIN {X 0,Y 418.271,Z 60.388,A -85,B 0,C 180,E1 -10140.895,E2 -10140.895} C_VEL
LIN {X 0,Y 418.377,Z 60.523,A -85,B 0,C 180,E1 -10142.003,E2 -10142.003} C_VEL
LIN {X 0,Y 420.883,Z 73.375,A -85,B 0,C 180,E1 -10144.567,E2 -10144.567} C_VEL
LIN {X 0,Y 420.896,Z 78.85,A -85,B 0,C 180,E1 -10145.589,E2 -10145.589} C_VEL
LIN {X 0,Y 420.004,Z 94.232,A -85,B 0,C 180,E1 -10148.399,E2 -10148.399} C_VEL
LIN {X 0,Y 419.156,Z 110.355,A -85,B 0,C 180,E1 -10151.32,E2 -10151.32} C_VEL
LIN {X 0,Y 422.902,Z 139.683,A -85,B 0,C 180,E1 -10151.974,E2 -10151.974} C_VEL
LIN {X 0,Y 422.015,Z 218.85,A -85,B 0,C 180,E1 -10153.336,E2 -10153.336} C_VEL
LIN {X 0,Y 421.566,Z 232.296,A -85,B 0,C 180,E1 -10153.754,E2 -10153.754} C_VEL
LIN {X 0,Y 421.002,Z 244.574,A -85,B 0,C 180,E1 -10154.322,E2 -10154.322} C_VEL
LIN {X 0,Y 420.261,Z 256.942,A -85,B 0,C 180,E1 -10155.101,E2 -10155.101} C_VEL
LIN {X 0,Y 419.558,Z 268.629,A -85,B 0,C 180,E1 -10156.066,E2 -10156.066} C_VEL
LIN {X 0,Y 418.939,Z 279.353,A -85,B 0,C 180,E1 -10157.179,E2 -10157.179} C_VEL
LIN {X 0,Y 418.362,Z 288.606,A -85,B 0,C 180,E1 -10158.37,E2 -10158.37} C_VEL
LIN {X 0,Y 417.731,Z 297.729,A -85,B 0,C 180,E1 -10159.825,E2 -10159.825} C_VEL
LIN {X 0,Y 417.426,Z 305.088,A -85,B 0,C 180,E1 -10161.284,E2 -10161.284} C_VEL
LIN {X 0,Y 417.241,Z 310.97,A -85,B 0,C 180,E1 -10162.742,E2 -10162.742} C_VEL
LIN {X 0,Y 417.067,Z 315.582,A -85,B 0,C 180,E1 -10164.197,E2 -10164.197} C_VEL
LIN {X 0,Y 417.133,Z 318.018,A -85,B 0,C 180,E1 -10165.167,E2 -10165.167} C_VEL
LIN {X 0,Y 417.07,Z 320.001,A -85,B 0,C 180,E1 -10166.135,E2 -10166.135} C_VEL
LIN {X 0,Y 417.167,Z 321.573,A -85,B 0,C 180,E1 -10167.103,E2 -10167.103} C_VEL
LIN {X 0,Y 417.137,Z 322.691,A -85,B 0,C 180,E1 -10168.069,E2 -10168.069} C_VEL
LIN {X 0,Y 417.118,Z 323.388,A -85,B 0,C 180,E1 -10169.034,E2 -10169.034} C_VEL
LIN {X 0,Y 417.12,Z 323.695,A -85,B 0,C 180,E1 -10170,E2 -10170} C_VEL
LIN {X 0,Y 417.092,Z 323.612,A -85,B 0,C 180,E1 -10170.965,E2 -10170.965} C_VEL
LIN {X 0,Y 417.118,Z 323.116,A -85,B 0,C 180,E1 -10171.931,E2 -10171.931} C_VEL
LIN {X 0,Y 417.129,Z 322.196,A -85,B 0,C 180,E1 -10172.897,E2 -10172.897} C_VEL
LIN {X 0,Y 417.099,Z 319.159,A -85,B 0,C 180,E1 -10174.832,E2 -10174.832} C_VEL
LIN {X 0,Y 417.05,Z 316.081,A -85,B 0,C 180,E1 -10176.146,E2 -10176.146} C_VEL
LIN {X 0,Y 417.307,Z 311.199,A -85,B 0,C 180,E1 -10177.743,E2 -10177.743} C_VEL
LIN {X 0,Y 417.647,Z 304.393,A -85,B 0,C 180,E1 -10179.443,E2 -10179.443} C_VEL
LIN {X 0,Y 418.156,Z 297.011,A -85,B 0,C 180,E1 -10180.899,E2 -10180.899} C_VEL
LIN {X 0,Y 418.945,Z 287.884,A -85,B 0,C 180,E1 -10182.35,E2 -10182.35} C_VEL
LIN {X 0,Y 419.621,Z 278.437,A -85,B 0,C 180,E1 -10183.56,E2 -10183.56} C_VEL
LIN {X 0,Y 420.493,Z 267.985,A -85,B 0,C 180,E1 -10184.643,E2 -10184.643} C_VEL
LIN {X 0,Y 421.331,Z 256.4,A -85,B 0,C 180,E1 -10185.603,E2 -10185.603} C_VEL
LIN {X 0,Y 422.252,Z 244.138,A -85,B 0,C 180,E1 -10186.374,E2 -10186.374} C_VEL
LIN {X 0,Y 422.996,Z 231.282,A -85,B 0,C 180,E1 -10186.965,E2 -10186.965} C_VEL
LIN {X 0,Y 423.548,Z 218.913,A -85,B 0,C 180,E1 -10187.347,E2 -10187.347} C_VEL
LIN {X 0,Y 424.474,Z 138.441,A -85,B 0,C 180,E1 -10188.765,E2 -10188.765} C_VEL
LIN {X 0,Y 421.734,Z 120.058,A -85,B 0,C 180,E1 -10189.243,E2 -10189.243} C_VEL
LIN {X 0,Y 419.888,Z 109.637,A -85,B 0,C 180,E1 -10189.557,E2 -10189.557} C_VEL
LIN {X 0,Y 420.961,Z 93.438,A -85,B 0,C 180,E1 -10192.581,E2 -10192.581} C_VEL
LIN {X 0,Y 422.007,Z 78.613,A -85,B 0,C 180,E1 -10195.393,E2 -10195.393} C_VEL
LIN {X 0,Y 420.909,Z 71.865,A -85,B 0,C 180,E1 -10196.796,E2 -10196.796} C_VEL
LIN {X 0,Y 418.248,Z 60.389,A -85,B 0,C 180,E1 -10199.335,E2 -10199.335} C_VEL
LIN {X 0,Y 418.257,Z 60.385,A -85,B 0,C 180,E1 -10202.844,E2 -10202.844} C_VEL
LIN {X 0,Y 418.248,Z 60.39,A -85,B 0,C 180,E1 -10206.238,E2 -10206.238} C_VEL
